// ============================================
// DB_RecipeProgram4 - SpinningCam Program
// Lines: 999
// Generated by SpinningCam  [2026-08-13 21:01:36]
// ============================================
//
// --- MAKINE AYARLARI ---
// Machine Origin  : X=0.0, Z=0.0
// Axis Direction  : X=NORMAL, Z=NORMAL
// Output Mode     : RADIUS
// G54 Offset      : X=0.0, Z=0.0
// Home            : X=-396.641, Z=-174.0
// Retract         : X=-10.0, Z=-10.0
//
// --- PARCA / BLANK ---
// Blank Radius    : 155.0 mm
// Blank Z Shift   : 0.0 mm
// Final Thickness : 0.8 mm
// Min Safety Gap  : 0.0 mm
//
// --- MANDREL POZISYON ---
// Mandrel Offset  : X=0.0, Z=0.0
// Mandrel Rot     : Rx=90.0, Ry=0.0, Rz=0.0
//
// --- OPERASYONLAR ---
// Op1: ROUGHING, 1 paso, T004, R=44.56mm, RPM=800.0, mm_min=800.0
// Op2: ROUGHING, 1 paso, T004, R=44.56mm, RPM=800.0, mm_min=800.0
// Op3: ROUGHING, 1 paso, T004, R=44.56mm, RPM=800.0, mm_min=800.0
// Op4: ROUGHING, 1 paso, T004, R=44.56mm, RPM=800.0, mm_min=800.0
// Op5: ROUGHING, 1 paso, T004, R=44.56mm, RPM=800.0, mm_min=800.0
// Op6: ROUGHING, 1 paso, T004, R=44.56mm, RPM=800.0, mm_min=500.0
// Op7: ROUGHING, 1 paso, T004, R=44.56mm, RPM=800.0, mm_min=500.0
// Op8: ROUGHING, 1 paso, T004, R=44.56mm, RPM=800.0, mm_min=800.0
// Op9: ROUGHING, 1 paso, T004, R=44.56mm, RPM=800.0, mm_min=800.0
// Op10: ROUGHING, 1 paso, T004, R=44.56mm, RPM=800.0, mm_min=800.0
// Op11: ROUGHING, 1 paso, T004, R=44.56mm, RPM=800.0, mm_min=800.0
// Op12: ROUGHING, 1 paso, T004, R=44.56mm, RPM=800.0, mm_min=800.0
// Op13: ROUGHING, 1 paso, T004, R=44.56mm, RPM=800.0, mm_min=400.0
// Op14: ROUGHING, 1 paso, T004, R=44.56mm, RPM=800.0, mm_min=400.0
// Op15: ROUGHING, 1 paso, T004, R=44.56mm, RPM=800.0, mm_min=400.0
// Op16: ROUGHING, 1 paso, T004, R=44.56mm, RPM=800.0, mm_min=400.0
// Op17: ROUGHING, 3 paso, T004, R=44.56mm, RPM=800.0, mm_min=400.0
// Op18: ROUGHING, 3 paso, T004, R=44.56mm, RPM=800.0, mm_min=400.0
// Op19: ROUGHING, 1 paso, T004, R=44.56mm, RPM=800.0, mm_min=800.0
// Op20: ROUGHING, 3 paso, T004, R=44.56mm, RPM=800.0, mm_min=400.0
// Op21: ROUGHING, 3 paso, T004, R=44.56mm, RPM=800.0, mm_min=400.0
// Op22: ROUGHING, 3 paso, T004, R=44.56mm, RPM=800.0, mm_min=400.0
// Op23: ROUGHING, 1 paso, T004, R=44.56mm, RPM=800.0, mm_min=400.0
// Op24: ROUGHING, 3 paso, T004, R=44.56mm, RPM=800.0, mm_min=400.0
// Op25: ROUGHING, 3 paso, T004, R=44.56mm, RPM=800.0, mm_min=400.0
// Op26: ROUGHING, 3 paso, T004, R=44.56mm, RPM=800.0, mm_min=400.0
// Op27: ROUGHING, 3 paso, T004, R=44.56mm, RPM=800.0, mm_min=400.0
// Op28: ROUGHING, 3 paso, T004, R=44.56mm, RPM=800.0, mm_min=400.0
// Op29: ROUGHING, 3 paso, T004, R=44.56mm, RPM=800.0, mm_min=400.0
// Op30: CUTTING, 1 paso, T0102, R=77.53mm, RPM=300.0, mm_min=50.0
// ============================================

DATA_BLOCK "DB_RecipeProgram4"
{ S7_Optimized_Access := 'FALSE' }
VERSION : 0.2
// UNLINKED restored 2026-08-13: the work-memory workaround is withdrawn, the
// chunked loader replaces it. This DB is back in load memory and costs no work
// memory. Its Lines array is declared in CHUNKS (Lines1..Lines10, 100 lines each)
// because READ_DBL can only point at a whole declared member -- see
// tools/split_recipe_db.py, which produced this layout from the CAM export.
UNLINKED
NON_RETAIN
    VAR
        Header : "RecipeHeader";
        Lines1 : Array[0..99] of "RecipeLine"; // global lines 0..99
        Lines2 : Array[0..99] of "RecipeLine"; // global lines 100..199
        Lines3 : Array[0..99] of "RecipeLine"; // global lines 200..299
        Lines4 : Array[0..99] of "RecipeLine"; // global lines 300..399
        Lines5 : Array[0..99] of "RecipeLine"; // global lines 400..499
        Lines6 : Array[0..99] of "RecipeLine"; // global lines 500..599
        Lines7 : Array[0..99] of "RecipeLine"; // global lines 600..699
        Lines8 : Array[0..99] of "RecipeLine"; // global lines 700..799
        Lines9 : Array[0..99] of "RecipeLine"; // global lines 800..899
        Lines10: Array[0..99] of "RecipeLine"; // global lines 900..999
    END_VAR
BEGIN
    // Header
    Header.sName := 'SpinningCam Program';
    Header.LineCount := 999;
    Header.Valid := TRUE;
    Header.PreScanned := FALSE;
    Header.MinX := 0.000;
    Header.MaxX := 275.949;
    Header.MinZ := 0.000;
    Header.MaxZ := 312.533;

    // --- Tool table (CAM-authored) ---
    Header.ProvidesToolConfig := TRUE;
    Header.ToolCount := 3;
    Header.AutoCalcAngles := FALSE;
    Header.ToolCode_List[1] := 4;
    Header.ToolCode_List[2] := 5;
    Header.ToolCode_List[3] := 6;
    Header.ToolCode_List[4] := 0;  // unused
    Header.ToolAngle_List[1] := 0.0;
    Header.ToolAngle_List[2] := 120.0;
    Header.ToolAngle_List[3] := 240.0;
    Header.ToolAngle_List[4] := 360.0;

    // Recipe Lines (999 total)
    Lines1[0].X := 0.000; Lines1[0].Z := 0.000; Lines1[0].F := 0; Lines1[0].CMD := 0; Lines1[0].Param := 0; // G0 Rapid
    Lines1[1].X := 0.000; Lines1[1].Z := 0.000; Lines1[1].F := 0; Lines1[1].CMD := 0; Lines1[1].Param := 0; // G0 Rapid
    Lines1[2].X := 0.000; Lines1[2].Z := 0.000; Lines1[2].F := 0; Lines1[2].CMD := 40; Lines1[2].Param := 80; // Cylinder GOTO 0 mm
    Lines1[3].X := 0.000; Lines1[3].Z := 0.000; Lines1[3].F := 0; Lines1[3].CMD := 10; Lines1[3].Param := 4; // Tool Change T4
    Lines1[4].X := 0.000; Lines1[4].Z := 0.000; Lines1[4].F := 0; Lines1[4].CMD := 20; Lines1[4].Param := 80; // Spindle ON 800 RPM
    Lines1[5].X := 0.000; Lines1[5].Z := 0.000; Lines1[5].F := 0; Lines1[5].CMD := 41; Lines1[5].Param := 1; // M41 (Clamp On) P1 [Op1 P1]
    Lines1[6].X := 275.742; Lines1[6].Z := 181.000; Lines1[6].F := 0; Lines1[6].CMD := 0; Lines1[6].Param := 0; // G0 Rapid [Op1 P1]
    Lines1[7].X := 275.736; Lines1[7].Z := 184.000; Lines1[7].F := 800; Lines1[7].CMD := 1; Lines1[7].Param := 0; // G1 Linear [Op1 P1]
    Lines1[8].X := 188.561; Lines1[8].Z := 203.393; Lines1[8].F := 800; Lines1[8].CMD := 1; Lines1[8].Param := 0; // G1 Linear [Op1 P1]
    Lines1[9].X := 178.561; Lines1[9].Z := 193.393; Lines1[9].F := 0; Lines1[9].CMD := 0; Lines1[9].Param := 0; // G0 Rapid [Op1 P1]
    Lines1[10].X := 178.561; Lines1[10].Z := 193.393; Lines1[10].F := 0; Lines1[10].CMD := 20; Lines1[10].Param := 80; // Spindle ON 800 RPM [Op1 P1]
    Lines1[11].X := 275.742; Lines1[11].Z := 182.538; Lines1[11].F := 0; Lines1[11].CMD := 0; Lines1[11].Param := 0; // G0 Rapid [Op2 P1]
    Lines1[12].X := 275.731; Lines1[12].Z := 185.538; Lines1[12].F := 800; Lines1[12].CMD := 1; Lines1[12].Param := 0; // G1 Linear [Op2 P1]
    Lines1[13].X := 185.741; Lines1[13].Z := 218.401; Lines1[13].F := 800; Lines1[13].CMD := 1; Lines1[13].Param := 0; // G1 Linear [Op2 P1]
    Lines1[14].X := 175.741; Lines1[14].Z := 208.401; Lines1[14].F := 0; Lines1[14].CMD := 0; Lines1[14].Param := 0; // G0 Rapid [Op2 P1]
    Lines1[15].X := 175.741; Lines1[15].Z := 208.401; Lines1[15].F := 0; Lines1[15].CMD := 20; Lines1[15].Param := 80; // Spindle ON 800 RPM [Op2 P1]
    Lines1[16].X := 275.747; Lines1[16].Z := 181.000; Lines1[16].F := 0; Lines1[16].CMD := 0; Lines1[16].Param := 0; // G0 Rapid [Op3 P1]
    Lines1[17].X := 275.718; Lines1[17].Z := 189.000; Lines1[17].F := 800; Lines1[17].CMD := 1; Lines1[17].Param := 0; // G1 Linear [Op3 P1]
    Lines1[18].X := 274.433; Lines1[18].Z := 189.804; Lines1[18].F := 800; Lines1[18].CMD := 1; Lines1[18].Param := 0; // G1 Linear [Op3 P1]
    Lines1[19].X := 273.146; Lines1[19].Z := 190.603; Lines1[19].F := 800; Lines1[19].CMD := 1; Lines1[19].Param := 0; // G1 Linear [Op3 P1]
    Lines1[20].X := 271.856; Lines1[20].Z := 191.396; Lines1[20].F := 800; Lines1[20].CMD := 1; Lines1[20].Param := 0; // G1 Linear [Op3 P1]
    Lines1[21].X := 270.563; Lines1[21].Z := 192.184; Lines1[21].F := 800; Lines1[21].CMD := 1; Lines1[21].Param := 0; // G1 Linear [Op3 P1]
    Lines1[22].X := 269.269; Lines1[22].Z := 192.967; Lines1[22].F := 800; Lines1[22].CMD := 1; Lines1[22].Param := 0; // G1 Linear [Op3 P1]
    Lines1[23].X := 267.971; Lines1[23].Z := 193.745; Lines1[23].F := 800; Lines1[23].CMD := 1; Lines1[23].Param := 0; // G1 Linear [Op3 P1]
    Lines1[24].X := 266.672; Lines1[24].Z := 194.517; Lines1[24].F := 800; Lines1[24].CMD := 1; Lines1[24].Param := 0; // G1 Linear [Op3 P1]
    Lines1[25].X := 265.370; Lines1[25].Z := 195.285; Lines1[25].F := 800; Lines1[25].CMD := 1; Lines1[25].Param := 0; // G1 Linear [Op3 P1]
    Lines1[26].X := 264.065; Lines1[26].Z := 196.047; Lines1[26].F := 800; Lines1[26].CMD := 1; Lines1[26].Param := 0; // G1 Linear [Op3 P1]
    Lines1[27].X := 262.758; Lines1[27].Z := 196.803; Lines1[27].F := 800; Lines1[27].CMD := 1; Lines1[27].Param := 0; // G1 Linear [Op3 P1]
    Lines1[28].X := 261.448; Lines1[28].Z := 197.555; Lines1[28].F := 800; Lines1[28].CMD := 1; Lines1[28].Param := 0; // G1 Linear [Op3 P1]
    Lines1[29].X := 260.136; Lines1[29].Z := 198.301; Lines1[29].F := 800; Lines1[29].CMD := 1; Lines1[29].Param := 0; // G1 Linear [Op3 P1]
    Lines1[30].X := 258.822; Lines1[30].Z := 199.042; Lines1[30].F := 800; Lines1[30].CMD := 1; Lines1[30].Param := 0; // G1 Linear [Op3 P1]
    Lines1[31].X := 257.505; Lines1[31].Z := 199.778; Lines1[31].F := 800; Lines1[31].CMD := 1; Lines1[31].Param := 0; // G1 Linear [Op3 P1]
    Lines1[32].X := 256.186; Lines1[32].Z := 200.508; Lines1[32].F := 800; Lines1[32].CMD := 1; Lines1[32].Param := 0; // G1 Linear [Op3 P1]
    Lines1[33].X := 254.864; Lines1[33].Z := 201.233; Lines1[33].F := 800; Lines1[33].CMD := 1; Lines1[33].Param := 0; // G1 Linear [Op3 P1]
    Lines1[34].X := 253.540; Lines1[34].Z := 201.953; Lines1[34].F := 800; Lines1[34].CMD := 1; Lines1[34].Param := 0; // G1 Linear [Op3 P1]
    Lines1[35].X := 252.213; Lines1[35].Z := 202.668; Lines1[35].F := 800; Lines1[35].CMD := 1; Lines1[35].Param := 0; // G1 Linear [Op3 P1]
    Lines1[36].X := 250.884; Lines1[36].Z := 203.377; Lines1[36].F := 800; Lines1[36].CMD := 1; Lines1[36].Param := 0; // G1 Linear [Op3 P1]
    Lines1[37].X := 249.552; Lines1[37].Z := 204.081; Lines1[37].F := 800; Lines1[37].CMD := 1; Lines1[37].Param := 0; // G1 Linear [Op3 P1]
    Lines1[38].X := 248.218; Lines1[38].Z := 204.780; Lines1[38].F := 800; Lines1[38].CMD := 1; Lines1[38].Param := 0; // G1 Linear [Op3 P1]
    Lines1[39].X := 246.881; Lines1[39].Z := 205.474; Lines1[39].F := 800; Lines1[39].CMD := 1; Lines1[39].Param := 0; // G1 Linear [Op3 P1]
    Lines1[40].X := 245.542; Lines1[40].Z := 206.162; Lines1[40].F := 800; Lines1[40].CMD := 1; Lines1[40].Param := 0; // G1 Linear [Op3 P1]
    Lines1[41].X := 244.201; Lines1[41].Z := 206.846; Lines1[41].F := 800; Lines1[41].CMD := 1; Lines1[41].Param := 0; // G1 Linear [Op3 P1]
    Lines1[42].X := 242.633; Lines1[42].Z := 207.636; Lines1[42].F := 800; Lines1[42].CMD := 1; Lines1[42].Param := 0; // G1 Linear [Op3 P1]
    Lines1[43].X := 241.286; Lines1[43].Z := 208.308; Lines1[43].F := 800; Lines1[43].CMD := 1; Lines1[43].Param := 0; // G1 Linear [Op3 P1]
    Lines1[44].X := 239.937; Lines1[44].Z := 208.974; Lines1[44].F := 800; Lines1[44].CMD := 1; Lines1[44].Param := 0; // G1 Linear [Op3 P1]
    Lines1[45].X := 238.585; Lines1[45].Z := 209.636; Lines1[45].F := 800; Lines1[45].CMD := 1; Lines1[45].Param := 0; // G1 Linear [Op3 P1]
    Lines1[46].X := 237.231; Lines1[46].Z := 210.292; Lines1[46].F := 800; Lines1[46].CMD := 1; Lines1[46].Param := 0; // G1 Linear [Op3 P1]
    Lines1[47].X := 235.874; Lines1[47].Z := 210.942; Lines1[47].F := 800; Lines1[47].CMD := 1; Lines1[47].Param := 0; // G1 Linear [Op3 P1]
    Lines1[48].X := 234.515; Lines1[48].Z := 211.588; Lines1[48].F := 800; Lines1[48].CMD := 1; Lines1[48].Param := 0; // G1 Linear [Op3 P1]
    Lines1[49].X := 233.154; Lines1[49].Z := 212.228; Lines1[49].F := 800; Lines1[49].CMD := 1; Lines1[49].Param := 0; // G1 Linear [Op3 P1]
    Lines1[50].X := 231.562; Lines1[50].Z := 212.969; Lines1[50].F := 800; Lines1[50].CMD := 1; Lines1[50].Param := 0; // G1 Linear [Op3 P1]
    Lines1[51].X := 230.195; Lines1[51].Z := 213.597; Lines1[51].F := 800; Lines1[51].CMD := 1; Lines1[51].Param := 0; // G1 Linear [Op3 P1]
    Lines1[52].X := 228.826; Lines1[52].Z := 214.221; Lines1[52].F := 800; Lines1[52].CMD := 1; Lines1[52].Param := 0; // G1 Linear [Op3 P1]
    Lines1[53].X := 227.454; Lines1[53].Z := 214.839; Lines1[53].F := 800; Lines1[53].CMD := 1; Lines1[53].Param := 0; // G1 Linear [Op3 P1]
    Lines1[54].X := 226.080; Lines1[54].Z := 215.453; Lines1[54].F := 800; Lines1[54].CMD := 1; Lines1[54].Param := 0; // G1 Linear [Op3 P1]
    Lines1[55].X := 224.703; Lines1[55].Z := 216.060; Lines1[55].F := 800; Lines1[55].CMD := 1; Lines1[55].Param := 0; // G1 Linear [Op3 P1]
    Lines1[56].X := 223.324; Lines1[56].Z := 216.663; Lines1[56].F := 800; Lines1[56].CMD := 1; Lines1[56].Param := 0; // G1 Linear [Op3 P1]
    Lines1[57].X := 221.942; Lines1[57].Z := 217.260; Lines1[57].F := 800; Lines1[57].CMD := 1; Lines1[57].Param := 0; // G1 Linear [Op3 P1]
    Lines1[58].X := 220.558; Lines1[58].Z := 217.853; Lines1[58].F := 800; Lines1[58].CMD := 1; Lines1[58].Param := 0; // G1 Linear [Op3 P1]
    Lines1[59].X := 219.172; Lines1[59].Z := 218.439; Lines1[59].F := 800; Lines1[59].CMD := 1; Lines1[59].Param := 0; // G1 Linear [Op3 P1]
    Lines1[60].X := 217.783; Lines1[60].Z := 219.021; Lines1[60].F := 800; Lines1[60].CMD := 1; Lines1[60].Param := 0; // G1 Linear [Op3 P1]
    Lines1[61].X := 216.391; Lines1[61].Z := 219.597; Lines1[61].F := 800; Lines1[61].CMD := 1; Lines1[61].Param := 0; // G1 Linear [Op3 P1]
    Lines1[62].X := 214.997; Lines1[62].Z := 220.169; Lines1[62].F := 800; Lines1[62].CMD := 1; Lines1[62].Param := 0; // G1 Linear [Op3 P1]
    Lines1[63].X := 213.601; Lines1[63].Z := 220.734; Lines1[63].F := 800; Lines1[63].CMD := 1; Lines1[63].Param := 0; // G1 Linear [Op3 P1]
    Lines1[64].X := 212.202; Lines1[64].Z := 221.295; Lines1[64].F := 800; Lines1[64].CMD := 1; Lines1[64].Param := 0; // G1 Linear [Op3 P1]
    Lines1[65].X := 210.801; Lines1[65].Z := 221.850; Lines1[65].F := 800; Lines1[65].CMD := 1; Lines1[65].Param := 0; // G1 Linear [Op3 P1]
    Lines1[66].X := 209.397; Lines1[66].Z := 222.401; Lines1[66].F := 800; Lines1[66].CMD := 1; Lines1[66].Param := 0; // G1 Linear [Op3 P1]
    Lines1[67].X := 207.991; Lines1[67].Z := 222.945; Lines1[67].F := 800; Lines1[67].CMD := 1; Lines1[67].Param := 0; // G1 Linear [Op3 P1]
    Lines1[68].X := 206.582; Lines1[68].Z := 223.485; Lines1[68].F := 800; Lines1[68].CMD := 1; Lines1[68].Param := 0; // G1 Linear [Op3 P1]
    Lines1[69].X := 205.171; Lines1[69].Z := 224.019; Lines1[69].F := 800; Lines1[69].CMD := 1; Lines1[69].Param := 0; // G1 Linear [Op3 P1]
    Lines1[70].X := 203.758; Lines1[70].Z := 224.548; Lines1[70].F := 800; Lines1[70].CMD := 1; Lines1[70].Param := 0; // G1 Linear [Op3 P1]
    Lines1[71].X := 202.342; Lines1[71].Z := 225.072; Lines1[71].F := 800; Lines1[71].CMD := 1; Lines1[71].Param := 0; // G1 Linear [Op3 P1]
    Lines1[72].X := 200.923; Lines1[72].Z := 225.591; Lines1[72].F := 800; Lines1[72].CMD := 1; Lines1[72].Param := 0; // G1 Linear [Op3 P1]
    Lines1[73].X := 199.502; Lines1[73].Z := 226.104; Lines1[73].F := 800; Lines1[73].CMD := 1; Lines1[73].Param := 0; // G1 Linear [Op3 P1]
    Lines1[74].X := 198.079; Lines1[74].Z := 226.612; Lines1[74].F := 800; Lines1[74].CMD := 1; Lines1[74].Param := 0; // G1 Linear [Op3 P1]
    Lines1[75].X := 196.653; Lines1[75].Z := 227.115; Lines1[75].F := 800; Lines1[75].CMD := 1; Lines1[75].Param := 0; // G1 Linear [Op3 P1]
    Lines1[76].X := 195.225; Lines1[76].Z := 227.613; Lines1[76].F := 800; Lines1[76].CMD := 1; Lines1[76].Param := 0; // G1 Linear [Op3 P1]
    Lines1[77].X := 193.794; Lines1[77].Z := 228.105; Lines1[77].F := 800; Lines1[77].CMD := 1; Lines1[77].Param := 0; // G1 Linear [Op3 P1]
    Lines1[78].X := 192.361; Lines1[78].Z := 228.592; Lines1[78].F := 800; Lines1[78].CMD := 1; Lines1[78].Param := 0; // G1 Linear [Op3 P1]
    Lines1[79].X := 190.925; Lines1[79].Z := 229.074; Lines1[79].F := 800; Lines1[79].CMD := 1; Lines1[79].Param := 0; // G1 Linear [Op3 P1]
    Lines1[80].X := 189.487; Lines1[80].Z := 229.551; Lines1[80].F := 800; Lines1[80].CMD := 1; Lines1[80].Param := 0; // G1 Linear [Op3 P1]
    Lines1[81].X := 188.046; Lines1[81].Z := 230.022; Lines1[81].F := 800; Lines1[81].CMD := 1; Lines1[81].Param := 0; // G1 Linear [Op3 P1]
    Lines1[82].X := 178.046; Lines1[82].Z := 220.022; Lines1[82].F := 0; Lines1[82].CMD := 0; Lines1[82].Param := 0; // G0 Rapid [Op3 P1]
    Lines1[83].X := 178.046; Lines1[83].Z := 220.022; Lines1[83].F := 0; Lines1[83].CMD := 20; Lines1[83].Param := 80; // Spindle ON 800 RPM [Op3 P1]
    Lines1[84].X := 275.747; Lines1[84].Z := 181.000; Lines1[84].F := 0; Lines1[84].CMD := 0; Lines1[84].Param := 0; // G0 Rapid [Op4 P1]
    Lines1[85].X := 275.703; Lines1[85].Z := 193.000; Lines1[85].F := 800; Lines1[85].CMD := 1; Lines1[85].Param := 0; // G1 Linear [Op4 P1]
    Lines1[86].X := 274.461; Lines1[86].Z := 193.867; Lines1[86].F := 800; Lines1[86].CMD := 1; Lines1[86].Param := 0; // G1 Linear [Op4 P1]
    Lines1[87].X := 273.215; Lines1[87].Z := 194.728; Lines1[87].F := 800; Lines1[87].CMD := 1; Lines1[87].Param := 0; // G1 Linear [Op4 P1]
    Lines1[88].X := 271.967; Lines1[88].Z := 195.585; Lines1[88].F := 800; Lines1[88].CMD := 1; Lines1[88].Param := 0; // G1 Linear [Op4 P1]
    Lines1[89].X := 270.508; Lines1[89].Z := 196.578; Lines1[89].F := 800; Lines1[89].CMD := 1; Lines1[89].Param := 0; // G1 Linear [Op4 P1]
    Lines1[90].X := 269.254; Lines1[90].Z := 197.425; Lines1[90].F := 800; Lines1[90].CMD := 1; Lines1[90].Param := 0; // G1 Linear [Op4 P1]
    Lines1[91].X := 267.998; Lines1[91].Z := 198.266; Lines1[91].F := 800; Lines1[91].CMD := 1; Lines1[91].Param := 0; // G1 Linear [Op4 P1]
    Lines1[92].X := 266.529; Lines1[92].Z := 199.241; Lines1[92].F := 800; Lines1[92].CMD := 1; Lines1[92].Param := 0; // G1 Linear [Op4 P1]
    Lines1[93].X := 265.267; Lines1[93].Z := 200.072; Lines1[93].F := 800; Lines1[93].CMD := 1; Lines1[93].Param := 0; // G1 Linear [Op4 P1]
    Lines1[94].X := 264.002; Lines1[94].Z := 200.898; Lines1[94].F := 800; Lines1[94].CMD := 1; Lines1[94].Param := 0; // G1 Linear [Op4 P1]
    Lines1[95].X := 262.735; Lines1[95].Z := 201.719; Lines1[95].F := 800; Lines1[95].CMD := 1; Lines1[95].Param := 0; // G1 Linear [Op4 P1]
    Lines1[96].X := 261.254; Lines1[96].Z := 202.670; Lines1[96].F := 800; Lines1[96].CMD := 1; Lines1[96].Param := 0; // G1 Linear [Op4 P1]
    Lines1[97].X := 259.981; Lines1[97].Z := 203.481; Lines1[97].F := 800; Lines1[97].CMD := 1; Lines1[97].Param := 0; // G1 Linear [Op4 P1]
    Lines1[98].X := 258.705; Lines1[98].Z := 204.286; Lines1[98].F := 800; Lines1[98].CMD := 1; Lines1[98].Param := 0; // G1 Linear [Op4 P1]
    Lines1[99].X := 257.427; Lines1[99].Z := 205.087; Lines1[99].F := 800; Lines1[99].CMD := 1; Lines1[99].Param := 0; // G1 Linear [Op4 P1]
    Lines2[0].X := 256.147; Lines2[0].Z := 205.882; Lines2[0].F := 800; Lines2[0].CMD := 1; Lines2[0].Param := 0; // G1 Linear [Op4 P1]
    Lines2[1].X := 254.864; Lines2[1].Z := 206.673; Lines2[1].F := 800; Lines2[1].CMD := 1; Lines2[1].Param := 0; // G1 Linear [Op4 P1]
    Lines2[2].X := 253.578; Lines2[2].Z := 207.459; Lines2[2].F := 800; Lines2[2].CMD := 1; Lines2[2].Param := 0; // G1 Linear [Op4 P1]
    Lines2[3].X := 252.074; Lines2[3].Z := 208.370; Lines2[3].F := 800; Lines2[3].CMD := 1; Lines2[3].Param := 0; // G1 Linear [Op4 P1]
    Lines2[4].X := 250.783; Lines2[4].Z := 209.145; Lines2[4].F := 800; Lines2[4].CMD := 1; Lines2[4].Param := 0; // G1 Linear [Op4 P1]
    Lines2[5].X := 249.489; Lines2[5].Z := 209.916; Lines2[5].F := 800; Lines2[5].CMD := 1; Lines2[5].Param := 0; // G1 Linear [Op4 P1]
    Lines2[6].X := 248.192; Lines2[6].Z := 210.681; Lines2[6].F := 800; Lines2[6].CMD := 1; Lines2[6].Param := 0; // G1 Linear [Op4 P1]
    Lines2[7].X := 246.676; Lines2[7].Z := 211.568; Lines2[7].F := 800; Lines2[7].CMD := 1; Lines2[7].Param := 0; // G1 Linear [Op4 P1]
    Lines2[8].X := 245.374; Lines2[8].Z := 212.323; Lines2[8].F := 800; Lines2[8].CMD := 1; Lines2[8].Param := 0; // G1 Linear [Op4 P1]
    Lines2[9].X := 244.069; Lines2[9].Z := 213.073; Lines2[9].F := 800; Lines2[9].CMD := 1; Lines2[9].Param := 0; // G1 Linear [Op4 P1]
    Lines2[10].X := 242.761; Lines2[10].Z := 213.819; Lines2[10].F := 800; Lines2[10].CMD := 1; Lines2[10].Param := 0; // G1 Linear [Op4 P1]
    Lines2[11].X := 241.451; Lines2[11].Z := 214.559; Lines2[11].F := 800; Lines2[11].CMD := 1; Lines2[11].Param := 0; // G1 Linear [Op4 P1]
    Lines2[12].X := 239.919; Lines2[12].Z := 215.417; Lines2[12].F := 800; Lines2[12].CMD := 1; Lines2[12].Param := 0; // G1 Linear [Op4 P1]
    Lines2[13].X := 238.603; Lines2[13].Z := 216.146; Lines2[13].F := 800; Lines2[13].CMD := 1; Lines2[13].Param := 0; // G1 Linear [Op4 P1]
    Lines2[14].X := 237.285; Lines2[14].Z := 216.871; Lines2[14].F := 800; Lines2[14].CMD := 1; Lines2[14].Param := 0; // G1 Linear [Op4 P1]
    Lines2[15].X := 235.964; Lines2[15].Z := 217.591; Lines2[15].F := 800; Lines2[15].CMD := 1; Lines2[15].Param := 0; // G1 Linear [Op4 P1]
    Lines2[16].X := 234.640; Lines2[16].Z := 218.306; Lines2[16].F := 800; Lines2[16].CMD := 1; Lines2[16].Param := 0; // G1 Linear [Op4 P1]
    Lines2[17].X := 233.314; Lines2[17].Z := 219.017; Lines2[17].F := 800; Lines2[17].CMD := 1; Lines2[17].Param := 0; // G1 Linear [Op4 P1]
    Lines2[18].X := 231.985; Lines2[18].Z := 219.722; Lines2[18].F := 800; Lines2[18].CMD := 1; Lines2[18].Param := 0; // G1 Linear [Op4 P1]
    Lines2[19].X := 230.654; Lines2[19].Z := 220.422; Lines2[19].F := 800; Lines2[19].CMD := 1; Lines2[19].Param := 0; // G1 Linear [Op4 P1]
    Lines2[20].X := 229.320; Lines2[20].Z := 221.118; Lines2[20].F := 800; Lines2[20].CMD := 1; Lines2[20].Param := 0; // G1 Linear [Op4 P1]
    Lines2[21].X := 227.760; Lines2[21].Z := 221.923; Lines2[21].F := 800; Lines2[21].CMD := 1; Lines2[21].Param := 0; // G1 Linear [Op4 P1]
    Lines2[22].X := 226.420; Lines2[22].Z := 222.608; Lines2[22].F := 800; Lines2[22].CMD := 1; Lines2[22].Param := 0; // G1 Linear [Op4 P1]
    Lines2[23].X := 225.078; Lines2[23].Z := 223.288; Lines2[23].F := 800; Lines2[23].CMD := 1; Lines2[23].Param := 0; // G1 Linear [Op4 P1]
    Lines2[24].X := 223.733; Lines2[24].Z := 223.963; Lines2[24].F := 800; Lines2[24].CMD := 1; Lines2[24].Param := 0; // G1 Linear [Op4 P1]
    Lines2[25].X := 222.386; Lines2[25].Z := 224.634; Lines2[25].F := 800; Lines2[25].CMD := 1; Lines2[25].Param := 0; // G1 Linear [Op4 P1]
    Lines2[26].X := 221.035; Lines2[26].Z := 225.299; Lines2[26].F := 800; Lines2[26].CMD := 1; Lines2[26].Param := 0; // G1 Linear [Op4 P1]
    Lines2[27].X := 219.683; Lines2[27].Z := 225.960; Lines2[27].F := 800; Lines2[27].CMD := 1; Lines2[27].Param := 0; // G1 Linear [Op4 P1]
    Lines2[28].X := 218.327; Lines2[28].Z := 226.615; Lines2[28].F := 800; Lines2[28].CMD := 1; Lines2[28].Param := 0; // G1 Linear [Op4 P1]
    Lines2[29].X := 216.969; Lines2[29].Z := 227.266; Lines2[29].F := 800; Lines2[29].CMD := 1; Lines2[29].Param := 0; // G1 Linear [Op4 P1]
    Lines2[30].X := 215.609; Lines2[30].Z := 227.912; Lines2[30].F := 800; Lines2[30].CMD := 1; Lines2[30].Param := 0; // G1 Linear [Op4 P1]
    Lines2[31].X := 214.018; Lines2[31].Z := 228.659; Lines2[31].F := 800; Lines2[31].CMD := 1; Lines2[31].Param := 0; // G1 Linear [Op4 P1]
    Lines2[32].X := 212.652; Lines2[32].Z := 229.295; Lines2[32].F := 800; Lines2[32].CMD := 1; Lines2[32].Param := 0; // G1 Linear [Op4 P1]
    Lines2[33].X := 211.283; Lines2[33].Z := 229.925; Lines2[33].F := 800; Lines2[33].CMD := 1; Lines2[33].Param := 0; // G1 Linear [Op4 P1]
    Lines2[34].X := 209.912; Lines2[34].Z := 230.550; Lines2[34].F := 800; Lines2[34].CMD := 1; Lines2[34].Param := 0; // G1 Linear [Op4 P1]
    Lines2[35].X := 208.538; Lines2[35].Z := 231.171; Lines2[35].F := 800; Lines2[35].CMD := 1; Lines2[35].Param := 0; // G1 Linear [Op4 P1]
    Lines2[36].X := 207.161; Lines2[36].Z := 231.787; Lines2[36].F := 800; Lines2[36].CMD := 1; Lines2[36].Param := 0; // G1 Linear [Op4 P1]
    Lines2[37].X := 205.782; Lines2[37].Z := 232.398; Lines2[37].F := 800; Lines2[37].CMD := 1; Lines2[37].Param := 0; // G1 Linear [Op4 P1]
    Lines2[38].X := 204.400; Lines2[38].Z := 233.004; Lines2[38].F := 800; Lines2[38].CMD := 1; Lines2[38].Param := 0; // G1 Linear [Op4 P1]
    Lines2[39].X := 202.785; Lines2[39].Z := 233.705; Lines2[39].F := 800; Lines2[39].CMD := 1; Lines2[39].Param := 0; // G1 Linear [Op4 P1]
    Lines2[40].X := 201.397; Lines2[40].Z := 234.300; Lines2[40].F := 800; Lines2[40].CMD := 1; Lines2[40].Param := 0; // G1 Linear [Op4 P1]
    Lines2[41].X := 200.007; Lines2[41].Z := 234.890; Lines2[41].F := 800; Lines2[41].CMD := 1; Lines2[41].Param := 0; // G1 Linear [Op4 P1]
    Lines2[42].X := 198.614; Lines2[42].Z := 235.476; Lines2[42].F := 800; Lines2[42].CMD := 1; Lines2[42].Param := 0; // G1 Linear [Op4 P1]
    Lines2[43].X := 196.986; Lines2[43].Z := 236.153; Lines2[43].F := 800; Lines2[43].CMD := 1; Lines2[43].Param := 0; // G1 Linear [Op4 P1]
    Lines2[44].X := 195.588; Lines2[44].Z := 236.728; Lines2[44].F := 800; Lines2[44].CMD := 1; Lines2[44].Param := 0; // G1 Linear [Op4 P1]
    Lines2[45].X := 194.187; Lines2[45].Z := 237.298; Lines2[45].F := 800; Lines2[45].CMD := 1; Lines2[45].Param := 0; // G1 Linear [Op4 P1]
    Lines2[46].X := 192.783; Lines2[46].Z := 237.864; Lines2[46].F := 800; Lines2[46].CMD := 1; Lines2[46].Param := 0; // G1 Linear [Op4 P1]
    Lines2[47].X := 191.377; Lines2[47].Z := 238.424; Lines2[47].F := 800; Lines2[47].CMD := 1; Lines2[47].Param := 0; // G1 Linear [Op4 P1]
    Lines2[48].X := 189.733; Lines2[48].Z := 239.072; Lines2[48].F := 800; Lines2[48].CMD := 1; Lines2[48].Param := 0; // G1 Linear [Op4 P1]
    Lines2[49].X := 188.321; Lines2[49].Z := 239.621; Lines2[49].F := 800; Lines2[49].CMD := 1; Lines2[49].Param := 0; // G1 Linear [Op4 P1]
    Lines2[50].X := 178.321; Lines2[50].Z := 229.621; Lines2[50].F := 0; Lines2[50].CMD := 0; Lines2[50].Param := 0; // G0 Rapid [Op4 P1]
    Lines2[51].X := 178.321; Lines2[51].Z := 229.621; Lines2[51].F := 0; Lines2[51].CMD := 20; Lines2[51].Param := 80; // Spindle ON 800 RPM [Op4 P1]
    Lines2[52].X := 275.447; Lines2[52].Z := 181.000; Lines2[52].F := 0; Lines2[52].CMD := 0; Lines2[52].Param := 0; // G0 Rapid [Op5 P1]
    Lines2[53].X := 275.389; Lines2[53].Z := 197.000; Lines2[53].F := 800; Lines2[53].CMD := 1; Lines2[53].Param := 0; // G1 Linear [Op5 P1]
    Lines2[54].X := 274.227; Lines2[54].Z := 197.972; Lines2[54].F := 800; Lines2[54].CMD := 1; Lines2[54].Param := 0; // G1 Linear [Op5 P1]
    Lines2[55].X := 273.062; Lines2[55].Z := 198.939; Lines2[55].F := 800; Lines2[55].CMD := 1; Lines2[55].Param := 0; // G1 Linear [Op5 P1]
    Lines2[56].X := 271.699; Lines2[56].Z := 200.062; Lines2[56].F := 800; Lines2[56].CMD := 1; Lines2[56].Param := 0; // G1 Linear [Op5 P1]
    Lines2[57].X := 270.528; Lines2[57].Z := 201.020; Lines2[57].F := 800; Lines2[57].CMD := 1; Lines2[57].Param := 0; // G1 Linear [Op5 P1]
    Lines2[58].X := 269.353; Lines2[58].Z := 201.973; Lines2[58].F := 800; Lines2[58].CMD := 1; Lines2[58].Param := 0; // G1 Linear [Op5 P1]
    Lines2[59].X := 267.980; Lines2[59].Z := 203.079; Lines2[59].F := 800; Lines2[59].CMD := 1; Lines2[59].Param := 0; // G1 Linear [Op5 P1]
    Lines2[60].X := 266.799; Lines2[60].Z := 204.022; Lines2[60].F := 800; Lines2[60].CMD := 1; Lines2[60].Param := 0; // G1 Linear [Op5 P1]
    Lines2[61].X := 265.615; Lines2[61].Z := 204.961; Lines2[61].F := 800; Lines2[61].CMD := 1; Lines2[61].Param := 0; // G1 Linear [Op5 P1]
    Lines2[62].X := 264.428; Lines2[62].Z := 205.895; Lines2[62].F := 800; Lines2[62].CMD := 1; Lines2[62].Param := 0; // G1 Linear [Op5 P1]
    Lines2[63].X := 263.239; Lines2[63].Z := 206.825; Lines2[63].F := 800; Lines2[63].CMD := 1; Lines2[63].Param := 0; // G1 Linear [Op5 P1]
    Lines2[64].X := 262.046; Lines2[64].Z := 207.750; Lines2[64].F := 800; Lines2[64].CMD := 1; Lines2[64].Param := 0; // G1 Linear [Op5 P1]
    Lines2[65].X := 260.651; Lines2[65].Z := 208.824; Lines2[65].F := 800; Lines2[65].CMD := 1; Lines2[65].Param := 0; // G1 Linear [Op5 P1]
    Lines2[66].X := 259.252; Lines2[66].Z := 209.891; Lines2[66].F := 800; Lines2[66].CMD := 1; Lines2[66].Param := 0; // G1 Linear [Op5 P1]
    Lines2[67].X := 258.050; Lines2[67].Z := 210.801; Lines2[67].F := 800; Lines2[67].CMD := 1; Lines2[67].Param := 0; // G1 Linear [Op5 P1]
    Lines2[68].X := 256.844; Lines2[68].Z := 211.707; Lines2[68].F := 800; Lines2[68].CMD := 1; Lines2[68].Param := 0; // G1 Linear [Op5 P1]
    Lines2[69].X := 255.636; Lines2[69].Z := 212.608; Lines2[69].F := 800; Lines2[69].CMD := 1; Lines2[69].Param := 0; // G1 Linear [Op5 P1]
    Lines2[70].X := 254.425; Lines2[70].Z := 213.504; Lines2[70].F := 800; Lines2[70].CMD := 1; Lines2[70].Param := 0; // G1 Linear [Op5 P1]
    Lines2[71].X := 253.211; Lines2[71].Z := 214.396; Lines2[71].F := 800; Lines2[71].CMD := 1; Lines2[71].Param := 0; // G1 Linear [Op5 P1]
    Lines2[72].X := 251.993; Lines2[72].Z := 215.284; Lines2[72].F := 800; Lines2[72].CMD := 1; Lines2[72].Param := 0; // G1 Linear [Op5 P1]
    Lines2[73].X := 250.570; Lines2[73].Z := 216.314; Lines2[73].F := 800; Lines2[73].CMD := 1; Lines2[73].Param := 0; // G1 Linear [Op5 P1]
    Lines2[74].X := 249.346; Lines2[74].Z := 217.191; Lines2[74].F := 800; Lines2[74].CMD := 1; Lines2[74].Param := 0; // G1 Linear [Op5 P1]
    Lines2[75].X := 248.119; Lines2[75].Z := 218.065; Lines2[75].F := 800; Lines2[75].CMD := 1; Lines2[75].Param := 0; // G1 Linear [Op5 P1]
    Lines2[76].X := 246.685; Lines2[76].Z := 219.078; Lines2[76].F := 800; Lines2[76].CMD := 1; Lines2[76].Param := 0; // G1 Linear [Op5 P1]
    Lines2[77].X := 245.452; Lines2[77].Z := 219.941; Lines2[77].F := 800; Lines2[77].CMD := 1; Lines2[77].Param := 0; // G1 Linear [Op5 P1]
    Lines2[78].X := 244.216; Lines2[78].Z := 220.800; Lines2[78].F := 800; Lines2[78].CMD := 1; Lines2[78].Param := 0; // G1 Linear [Op5 P1]
    Lines2[79].X := 242.977; Lines2[79].Z := 221.654; Lines2[79].F := 800; Lines2[79].CMD := 1; Lines2[79].Param := 0; // G1 Linear [Op5 P1]
    Lines2[80].X := 241.528; Lines2[80].Z := 222.645; Lines2[80].F := 800; Lines2[80].CMD := 1; Lines2[80].Param := 0; // G1 Linear [Op5 P1]
    Lines2[81].X := 240.283; Lines2[81].Z := 223.490; Lines2[81].F := 800; Lines2[81].CMD := 1; Lines2[81].Param := 0; // G1 Linear [Op5 P1]
    Lines2[82].X := 239.034; Lines2[82].Z := 224.330; Lines2[82].F := 800; Lines2[82].CMD := 1; Lines2[82].Param := 0; // G1 Linear [Op5 P1]
    Lines2[83].X := 237.783; Lines2[83].Z := 225.165; Lines2[83].F := 800; Lines2[83].CMD := 1; Lines2[83].Param := 0; // G1 Linear [Op5 P1]
    Lines2[84].X := 236.320; Lines2[84].Z := 226.135; Lines2[84].F := 800; Lines2[84].CMD := 1; Lines2[84].Param := 0; // G1 Linear [Op5 P1]
    Lines2[85].X := 235.062; Lines2[85].Z := 226.960; Lines2[85].F := 800; Lines2[85].CMD := 1; Lines2[85].Param := 0; // G1 Linear [Op5 P1]
    Lines2[86].X := 233.802; Lines2[86].Z := 227.782; Lines2[86].F := 800; Lines2[86].CMD := 1; Lines2[86].Param := 0; // G1 Linear [Op5 P1]
    Lines2[87].X := 232.538; Lines2[87].Z := 228.598; Lines2[87].F := 800; Lines2[87].CMD := 1; Lines2[87].Param := 0; // G1 Linear [Op5 P1]
    Lines2[88].X := 231.272; Lines2[88].Z := 229.410; Lines2[88].F := 800; Lines2[88].CMD := 1; Lines2[88].Param := 0; // G1 Linear [Op5 P1]
    Lines2[89].X := 229.791; Lines2[89].Z := 230.352; Lines2[89].F := 800; Lines2[89].CMD := 1; Lines2[89].Param := 0; // G1 Linear [Op5 P1]
    Lines2[90].X := 228.518; Lines2[90].Z := 231.155; Lines2[90].F := 800; Lines2[90].CMD := 1; Lines2[90].Param := 0; // G1 Linear [Op5 P1]
    Lines2[91].X := 227.242; Lines2[91].Z := 231.953; Lines2[91].F := 800; Lines2[91].CMD := 1; Lines2[91].Param := 0; // G1 Linear [Op5 P1]
    Lines2[92].X := 225.963; Lines2[92].Z := 232.746; Lines2[92].F := 800; Lines2[92].CMD := 1; Lines2[92].Param := 0; // G1 Linear [Op5 P1]
    Lines2[93].X := 224.467; Lines2[93].Z := 233.666; Lines2[93].F := 800; Lines2[93].CMD := 1; Lines2[93].Param := 0; // G1 Linear [Op5 P1]
    Lines2[94].X := 223.182; Lines2[94].Z := 234.449; Lines2[94].F := 800; Lines2[94].CMD := 1; Lines2[94].Param := 0; // G1 Linear [Op5 P1]
    Lines2[95].X := 221.894; Lines2[95].Z := 235.228; Lines2[95].F := 800; Lines2[95].CMD := 1; Lines2[95].Param := 0; // G1 Linear [Op5 P1]
    Lines2[96].X := 220.603; Lines2[96].Z := 236.003; Lines2[96].F := 800; Lines2[96].CMD := 1; Lines2[96].Param := 0; // G1 Linear [Op5 P1]
    Lines2[97].X := 219.093; Lines2[97].Z := 236.901; Lines2[97].F := 800; Lines2[97].CMD := 1; Lines2[97].Param := 0; // G1 Linear [Op5 P1]
    Lines2[98].X := 217.796; Lines2[98].Z := 237.666; Lines2[98].F := 800; Lines2[98].CMD := 1; Lines2[98].Param := 0; // G1 Linear [Op5 P1]
    Lines2[99].X := 216.495; Lines2[99].Z := 238.426; Lines2[99].F := 800; Lines2[99].CMD := 1; Lines2[99].Param := 0; // G1 Linear [Op5 P1]
    Lines3[0].X := 215.192; Lines3[0].Z := 239.181; Lines3[0].F := 800; Lines3[0].CMD := 1; Lines3[0].Param := 0; // G1 Linear [Op5 P1]
    Lines3[1].X := 213.667; Lines3[1].Z := 240.057; Lines3[1].F := 800; Lines3[1].CMD := 1; Lines3[1].Param := 0; // G1 Linear [Op5 P1]
    Lines3[2].X := 212.358; Lines3[2].Z := 240.803; Lines3[2].F := 800; Lines3[2].CMD := 1; Lines3[2].Param := 0; // G1 Linear [Op5 P1]
    Lines3[3].X := 211.045; Lines3[3].Z := 241.545; Lines3[3].F := 800; Lines3[3].CMD := 1; Lines3[3].Param := 0; // G1 Linear [Op5 P1]
    Lines3[4].X := 209.729; Lines3[4].Z := 242.282; Lines3[4].F := 800; Lines3[4].CMD := 1; Lines3[4].Param := 0; // G1 Linear [Op5 P1]
    Lines3[5].X := 208.190; Lines3[5].Z := 243.136; Lines3[5].F := 800; Lines3[5].CMD := 1; Lines3[5].Param := 0; // G1 Linear [Op5 P1]
    Lines3[6].X := 206.868; Lines3[6].Z := 243.863; Lines3[6].F := 800; Lines3[6].CMD := 1; Lines3[6].Param := 0; // G1 Linear [Op5 P1]
    Lines3[7].X := 205.322; Lines3[7].Z := 244.705; Lines3[7].F := 800; Lines3[7].CMD := 1; Lines3[7].Param := 0; // G1 Linear [Op5 P1]
    Lines3[8].X := 203.994; Lines3[8].Z := 245.422; Lines3[8].F := 800; Lines3[8].CMD := 1; Lines3[8].Param := 0; // G1 Linear [Op5 P1]
    Lines3[9].X := 202.662; Lines3[9].Z := 246.135; Lines3[9].F := 800; Lines3[9].CMD := 1; Lines3[9].Param := 0; // G1 Linear [Op5 P1]
    Lines3[10].X := 201.328; Lines3[10].Z := 246.844; Lines3[10].F := 800; Lines3[10].CMD := 1; Lines3[10].Param := 0; // G1 Linear [Op5 P1]
    Lines3[11].X := 199.990; Lines3[11].Z := 247.547; Lines3[11].F := 800; Lines3[11].CMD := 1; Lines3[11].Param := 0; // G1 Linear [Op5 P1]
    Lines3[12].X := 198.650; Lines3[12].Z := 248.246; Lines3[12].F := 800; Lines3[12].CMD := 1; Lines3[12].Param := 0; // G1 Linear [Op5 P1]
    Lines3[13].X := 197.082; Lines3[13].Z := 249.056; Lines3[13].F := 800; Lines3[13].CMD := 1; Lines3[13].Param := 0; // G1 Linear [Op5 P1]
    Lines3[14].X := 195.736; Lines3[14].Z := 249.746; Lines3[14].F := 800; Lines3[14].CMD := 1; Lines3[14].Param := 0; // G1 Linear [Op5 P1]
    Lines3[15].X := 194.386; Lines3[15].Z := 250.431; Lines3[15].F := 800; Lines3[15].CMD := 1; Lines3[15].Param := 0; // G1 Linear [Op5 P1]
    Lines3[16].X := 193.033; Lines3[16].Z := 251.111; Lines3[16].F := 800; Lines3[16].CMD := 1; Lines3[16].Param := 0; // G1 Linear [Op5 P1]
    Lines3[17].X := 191.451; Lines3[17].Z := 251.899; Lines3[17].F := 800; Lines3[17].CMD := 1; Lines3[17].Param := 0; // G1 Linear [Op5 P1]
    Lines3[18].X := 192.808; Lines3[18].Z := 251.224; Lines3[18].F := 800; Lines3[18].CMD := 1; Lines3[18].Param := 0; // G1 Linear [Op5 P1]
    Lines3[19].X := 194.161; Lines3[19].Z := 250.545; Lines3[19].F := 800; Lines3[19].CMD := 1; Lines3[19].Param := 0; // G1 Linear [Op5 P1]
    Lines3[20].X := 195.736; Lines3[20].Z := 249.746; Lines3[20].F := 800; Lines3[20].CMD := 1; Lines3[20].Param := 0; // G1 Linear [Op5 P1]
    Lines3[21].X := 197.082; Lines3[21].Z := 249.056; Lines3[21].F := 800; Lines3[21].CMD := 1; Lines3[21].Param := 0; // G1 Linear [Op5 P1]
    Lines3[22].X := 198.426; Lines3[22].Z := 248.363; Lines3[22].F := 800; Lines3[22].CMD := 1; Lines3[22].Param := 0; // G1 Linear [Op5 P1]
    Lines3[23].X := 199.990; Lines3[23].Z := 247.547; Lines3[23].F := 800; Lines3[23].CMD := 1; Lines3[23].Param := 0; // G1 Linear [Op5 P1]
    Lines3[24].X := 201.328; Lines3[24].Z := 246.844; Lines3[24].F := 800; Lines3[24].CMD := 1; Lines3[24].Param := 0; // G1 Linear [Op5 P1]
    Lines3[25].X := 202.662; Lines3[25].Z := 246.135; Lines3[25].F := 800; Lines3[25].CMD := 1; Lines3[25].Param := 0; // G1 Linear [Op5 P1]
    Lines3[26].X := 203.994; Lines3[26].Z := 245.422; Lines3[26].F := 800; Lines3[26].CMD := 1; Lines3[26].Param := 0; // G1 Linear [Op5 P1]
    Lines3[27].X := 205.322; Lines3[27].Z := 244.705; Lines3[27].F := 800; Lines3[27].CMD := 1; Lines3[27].Param := 0; // G1 Linear [Op5 P1]
    Lines3[28].X := 206.648; Lines3[28].Z := 243.983; Lines3[28].F := 800; Lines3[28].CMD := 1; Lines3[28].Param := 0; // G1 Linear [Op5 P1]
    Lines3[29].X := 208.190; Lines3[29].Z := 243.136; Lines3[29].F := 800; Lines3[29].CMD := 1; Lines3[29].Param := 0; // G1 Linear [Op5 P1]
    Lines3[30].X := 209.510; Lines3[30].Z := 242.404; Lines3[30].F := 800; Lines3[30].CMD := 1; Lines3[30].Param := 0; // G1 Linear [Op5 P1]
    Lines3[31].X := 210.826; Lines3[31].Z := 241.668; Lines3[31].F := 800; Lines3[31].CMD := 1; Lines3[31].Param := 0; // G1 Linear [Op5 P1]
    Lines3[32].X := 212.139; Lines3[32].Z := 240.927; Lines3[32].F := 800; Lines3[32].CMD := 1; Lines3[32].Param := 0; // G1 Linear [Op5 P1]
    Lines3[33].X := 213.667; Lines3[33].Z := 240.057; Lines3[33].F := 800; Lines3[33].CMD := 1; Lines3[33].Param := 0; // G1 Linear [Op5 P1]
    Lines3[34].X := 214.974; Lines3[34].Z := 239.307; Lines3[34].F := 800; Lines3[34].CMD := 1; Lines3[34].Param := 0; // G1 Linear [Op5 P1]
    Lines3[35].X := 216.278; Lines3[35].Z := 238.552; Lines3[35].F := 800; Lines3[35].CMD := 1; Lines3[35].Param := 0; // G1 Linear [Op5 P1]
    Lines3[36].X := 217.796; Lines3[36].Z := 237.666; Lines3[36].F := 800; Lines3[36].CMD := 1; Lines3[36].Param := 0; // G1 Linear [Op5 P1]
    Lines3[37].X := 219.093; Lines3[37].Z := 236.901; Lines3[37].F := 800; Lines3[37].CMD := 1; Lines3[37].Param := 0; // G1 Linear [Op5 P1]
    Lines3[38].X := 220.603; Lines3[38].Z := 236.003; Lines3[38].F := 800; Lines3[38].CMD := 1; Lines3[38].Param := 0; // G1 Linear [Op5 P1]
    Lines3[39].X := 221.894; Lines3[39].Z := 235.228; Lines3[39].F := 800; Lines3[39].CMD := 1; Lines3[39].Param := 0; // G1 Linear [Op5 P1]
    Lines3[40].X := 223.182; Lines3[40].Z := 234.449; Lines3[40].F := 800; Lines3[40].CMD := 1; Lines3[40].Param := 0; // G1 Linear [Op5 P1]
    Lines3[41].X := 224.467; Lines3[41].Z := 233.666; Lines3[41].F := 800; Lines3[41].CMD := 1; Lines3[41].Param := 0; // G1 Linear [Op5 P1]
    Lines3[42].X := 225.750; Lines3[42].Z := 232.878; Lines3[42].F := 800; Lines3[42].CMD := 1; Lines3[42].Param := 0; // G1 Linear [Op5 P1]
    Lines3[43].X := 227.029; Lines3[43].Z := 232.085; Lines3[43].F := 800; Lines3[43].CMD := 1; Lines3[43].Param := 0; // G1 Linear [Op5 P1]
    Lines3[44].X := 228.518; Lines3[44].Z := 231.155; Lines3[44].F := 800; Lines3[44].CMD := 1; Lines3[44].Param := 0; // G1 Linear [Op5 P1]
    Lines3[45].X := 229.791; Lines3[45].Z := 230.352; Lines3[45].F := 800; Lines3[45].CMD := 1; Lines3[45].Param := 0; // G1 Linear [Op5 P1]
    Lines3[46].X := 231.060; Lines3[46].Z := 229.545; Lines3[46].F := 800; Lines3[46].CMD := 1; Lines3[46].Param := 0; // G1 Linear [Op5 P1]
    Lines3[47].X := 232.327; Lines3[47].Z := 228.734; Lines3[47].F := 800; Lines3[47].CMD := 1; Lines3[47].Param := 0; // G1 Linear [Op5 P1]
    Lines3[48].X := 233.802; Lines3[48].Z := 227.782; Lines3[48].F := 800; Lines3[48].CMD := 1; Lines3[48].Param := 0; // G1 Linear [Op5 P1]
    Lines3[49].X := 235.062; Lines3[49].Z := 226.960; Lines3[49].F := 800; Lines3[49].CMD := 1; Lines3[49].Param := 0; // G1 Linear [Op5 P1]
    Lines3[50].X := 236.320; Lines3[50].Z := 226.135; Lines3[50].F := 800; Lines3[50].CMD := 1; Lines3[50].Param := 0; // G1 Linear [Op5 P1]
    Lines3[51].X := 237.783; Lines3[51].Z := 225.165; Lines3[51].F := 800; Lines3[51].CMD := 1; Lines3[51].Param := 0; // G1 Linear [Op5 P1]
    Lines3[52].X := 239.034; Lines3[52].Z := 224.330; Lines3[52].F := 800; Lines3[52].CMD := 1; Lines3[52].Param := 0; // G1 Linear [Op5 P1]
    Lines3[53].X := 240.283; Lines3[53].Z := 223.490; Lines3[53].F := 800; Lines3[53].CMD := 1; Lines3[53].Param := 0; // G1 Linear [Op5 P1]
    Lines3[54].X := 241.528; Lines3[54].Z := 222.645; Lines3[54].F := 800; Lines3[54].CMD := 1; Lines3[54].Param := 0; // G1 Linear [Op5 P1]
    Lines3[55].X := 242.977; Lines3[55].Z := 221.654; Lines3[55].F := 800; Lines3[55].CMD := 1; Lines3[55].Param := 0; // G1 Linear [Op5 P1]
    Lines3[56].X := 244.216; Lines3[56].Z := 220.800; Lines3[56].F := 800; Lines3[56].CMD := 1; Lines3[56].Param := 0; // G1 Linear [Op5 P1]
    Lines3[57].X := 245.452; Lines3[57].Z := 219.941; Lines3[57].F := 800; Lines3[57].CMD := 1; Lines3[57].Param := 0; // G1 Linear [Op5 P1]
    Lines3[58].X := 246.685; Lines3[58].Z := 219.078; Lines3[58].F := 800; Lines3[58].CMD := 1; Lines3[58].Param := 0; // G1 Linear [Op5 P1]
    Lines3[59].X := 248.119; Lines3[59].Z := 218.065; Lines3[59].F := 800; Lines3[59].CMD := 1; Lines3[59].Param := 0; // G1 Linear [Op5 P1]
    Lines3[60].X := 249.346; Lines3[60].Z := 217.191; Lines3[60].F := 800; Lines3[60].CMD := 1; Lines3[60].Param := 0; // G1 Linear [Op5 P1]
    Lines3[61].X := 250.570; Lines3[61].Z := 216.314; Lines3[61].F := 800; Lines3[61].CMD := 1; Lines3[61].Param := 0; // G1 Linear [Op5 P1]
    Lines3[62].X := 251.790; Lines3[62].Z := 215.431; Lines3[62].F := 800; Lines3[62].CMD := 1; Lines3[62].Param := 0; // G1 Linear [Op5 P1]
    Lines3[63].X := 253.211; Lines3[63].Z := 214.396; Lines3[63].F := 800; Lines3[63].CMD := 1; Lines3[63].Param := 0; // G1 Linear [Op5 P1]
    Lines3[64].X := 254.425; Lines3[64].Z := 213.504; Lines3[64].F := 800; Lines3[64].CMD := 1; Lines3[64].Param := 0; // G1 Linear [Op5 P1]
    Lines3[65].X := 255.636; Lines3[65].Z := 212.608; Lines3[65].F := 800; Lines3[65].CMD := 1; Lines3[65].Param := 0; // G1 Linear [Op5 P1]
    Lines3[66].X := 256.844; Lines3[66].Z := 211.707; Lines3[66].F := 800; Lines3[66].CMD := 1; Lines3[66].Param := 0; // G1 Linear [Op5 P1]
    Lines3[67].X := 258.050; Lines3[67].Z := 210.801; Lines3[67].F := 800; Lines3[67].CMD := 1; Lines3[67].Param := 0; // G1 Linear [Op5 P1]
    Lines3[68].X := 259.252; Lines3[68].Z := 209.891; Lines3[68].F := 800; Lines3[68].CMD := 1; Lines3[68].Param := 0; // G1 Linear [Op5 P1]
    Lines3[69].X := 260.651; Lines3[69].Z := 208.824; Lines3[69].F := 800; Lines3[69].CMD := 1; Lines3[69].Param := 0; // G1 Linear [Op5 P1]
    Lines3[70].X := 261.847; Lines3[70].Z := 207.904; Lines3[70].F := 800; Lines3[70].CMD := 1; Lines3[70].Param := 0; // G1 Linear [Op5 P1]
    Lines3[71].X := 263.239; Lines3[71].Z := 206.825; Lines3[71].F := 800; Lines3[71].CMD := 1; Lines3[71].Param := 0; // G1 Linear [Op5 P1]
    Lines3[72].X := 264.428; Lines3[72].Z := 205.895; Lines3[72].F := 800; Lines3[72].CMD := 1; Lines3[72].Param := 0; // G1 Linear [Op5 P1]
    Lines3[73].X := 265.615; Lines3[73].Z := 204.961; Lines3[73].F := 800; Lines3[73].CMD := 1; Lines3[73].Param := 0; // G1 Linear [Op5 P1]
    Lines3[74].X := 266.799; Lines3[74].Z := 204.022; Lines3[74].F := 800; Lines3[74].CMD := 1; Lines3[74].Param := 0; // G1 Linear [Op5 P1]
    Lines3[75].X := 267.980; Lines3[75].Z := 203.079; Lines3[75].F := 800; Lines3[75].CMD := 1; Lines3[75].Param := 0; // G1 Linear [Op5 P1]
    Lines3[76].X := 269.353; Lines3[76].Z := 201.973; Lines3[76].F := 800; Lines3[76].CMD := 1; Lines3[76].Param := 0; // G1 Linear [Op5 P1]
    Lines3[77].X := 270.528; Lines3[77].Z := 201.020; Lines3[77].F := 800; Lines3[77].CMD := 1; Lines3[77].Param := 0; // G1 Linear [Op5 P1]
    Lines3[78].X := 271.699; Lines3[78].Z := 200.062; Lines3[78].F := 800; Lines3[78].CMD := 1; Lines3[78].Param := 0; // G1 Linear [Op5 P1]
    Lines3[79].X := 273.062; Lines3[79].Z := 198.939; Lines3[79].F := 800; Lines3[79].CMD := 1; Lines3[79].Param := 0; // G1 Linear [Op5 P1]
    Lines3[80].X := 274.227; Lines3[80].Z := 197.972; Lines3[80].F := 800; Lines3[80].CMD := 1; Lines3[80].Param := 0; // G1 Linear [Op5 P1]
    Lines3[81].X := 275.389; Lines3[81].Z := 197.000; Lines3[81].F := 800; Lines3[81].CMD := 1; Lines3[81].Param := 0; // G1 Linear [Op5 P1]
    Lines3[82].X := 265.389; Lines3[82].Z := 187.000; Lines3[82].F := 0; Lines3[82].CMD := 0; Lines3[82].Param := 0; // G0 Rapid [Op5 P1]
    Lines3[83].X := 265.389; Lines3[83].Z := 187.000; Lines3[83].F := 0; Lines3[83].CMD := 20; Lines3[83].Param := 80; // Spindle ON 800 RPM [Op5 P1]
    Lines3[84].X := 275.449; Lines3[84].Z := 181.000; Lines3[84].F := 0; Lines3[84].CMD := 0; Lines3[84].Param := 0; // G0 Rapid [Op6 P1]
    Lines3[85].X := 275.382; Lines3[85].Z := 201.000; Lines3[85].F := 500; Lines3[85].CMD := 1; Lines3[85].Param := 0; // G1 Linear [Op6 P1]
    Lines3[86].X := 274.126; Lines3[86].Z := 202.242; Lines3[86].F := 500; Lines3[86].CMD := 1; Lines3[86].Param := 0; // G1 Linear [Op6 P1]
    Lines3[87].X := 273.046; Lines3[87].Z := 203.302; Lines3[87].F := 500; Lines3[87].CMD := 1; Lines3[87].Param := 0; // G1 Linear [Op6 P1]
    Lines3[88].X := 271.782; Lines3[88].Z := 204.534; Lines3[88].F := 500; Lines3[88].CMD := 1; Lines3[88].Param := 0; // G1 Linear [Op6 P1]
    Lines3[89].X := 270.695; Lines3[89].Z := 205.586; Lines3[89].F := 500; Lines3[89].CMD := 1; Lines3[89].Param := 0; // G1 Linear [Op6 P1]
    Lines3[90].X := 269.605; Lines3[90].Z := 206.633; Lines3[90].F := 500; Lines3[90].CMD := 1; Lines3[90].Param := 0; // G1 Linear [Op6 P1]
    Lines3[91].X := 268.329; Lines3[91].Z := 207.851; Lines3[91].F := 500; Lines3[91].CMD := 1; Lines3[91].Param := 0; // G1 Linear [Op6 P1]
    Lines3[92].X := 267.050; Lines3[92].Z := 209.063; Lines3[92].F := 500; Lines3[92].CMD := 1; Lines3[92].Param := 0; // G1 Linear [Op6 P1]
    Lines3[93].X := 265.949; Lines3[93].Z := 210.097; Lines3[93].F := 500; Lines3[93].CMD := 1; Lines3[93].Param := 0; // G1 Linear [Op6 P1]
    Lines3[94].X := 264.662; Lines3[94].Z := 211.300; Lines3[94].F := 500; Lines3[94].CMD := 1; Lines3[94].Param := 0; // G1 Linear [Op6 P1]
    Lines3[95].X := 263.555; Lines3[95].Z := 212.326; Lines3[95].F := 500; Lines3[95].CMD := 1; Lines3[95].Param := 0; // G1 Linear [Op6 P1]
    Lines3[96].X := 262.259; Lines3[96].Z := 213.518; Lines3[96].F := 500; Lines3[96].CMD := 1; Lines3[96].Param := 0; // G1 Linear [Op6 P1]
    Lines3[97].X := 261.145; Lines3[97].Z := 214.535; Lines3[97].F := 500; Lines3[97].CMD := 1; Lines3[97].Param := 0; // G1 Linear [Op6 P1]
    Lines3[98].X := 259.842; Lines3[98].Z := 215.717; Lines3[98].F := 500; Lines3[98].CMD := 1; Lines3[98].Param := 0; // G1 Linear [Op6 P1]
    Lines3[99].X := 258.722; Lines3[99].Z := 216.726; Lines3[99].F := 500; Lines3[99].CMD := 1; Lines3[99].Param := 0; // G1 Linear [Op6 P1]
    Lines4[0].X := 257.598; Lines4[0].Z := 217.731; Lines4[0].F := 500; Lines4[0].CMD := 1; Lines4[0].Param := 0; // G1 Linear [Op6 P1]
    Lines4[1].X := 256.283; Lines4[1].Z := 218.899; Lines4[1].F := 500; Lines4[1].CMD := 1; Lines4[1].Param := 0; // G1 Linear [Op6 P1]
    Lines4[2].X := 255.153; Lines4[2].Z := 219.895; Lines4[2].F := 500; Lines4[2].CMD := 1; Lines4[2].Param := 0; // G1 Linear [Op6 P1]
    Lines4[3].X := 253.831; Lines4[3].Z := 221.053; Lines4[3].F := 500; Lines4[3].CMD := 1; Lines4[3].Param := 0; // G1 Linear [Op6 P1]
    Lines4[4].X := 252.694; Lines4[4].Z := 222.041; Lines4[4].F := 500; Lines4[4].CMD := 1; Lines4[4].Param := 0; // G1 Linear [Op6 P1]
    Lines4[5].X := 251.363; Lines4[5].Z := 223.189; Lines4[5].F := 500; Lines4[5].CMD := 1; Lines4[5].Param := 0; // G1 Linear [Op6 P1]
    Lines4[6].X := 250.219; Lines4[6].Z := 224.168; Lines4[6].F := 500; Lines4[6].CMD := 1; Lines4[6].Param := 0; // G1 Linear [Op6 P1]
    Lines4[7].X := 248.881; Lines4[7].Z := 225.306; Lines4[7].F := 500; Lines4[7].CMD := 1; Lines4[7].Param := 0; // G1 Linear [Op6 P1]
    Lines4[8].X := 247.539; Lines4[8].Z := 226.438; Lines4[8].F := 500; Lines4[8].CMD := 1; Lines4[8].Param := 0; // G1 Linear [Op6 P1]
    Lines4[9].X := 246.384; Lines4[9].Z := 227.404; Lines4[9].F := 500; Lines4[9].CMD := 1; Lines4[9].Param := 0; // G1 Linear [Op6 P1]
    Lines4[10].X := 245.227; Lines4[10].Z := 228.366; Lines4[10].F := 500; Lines4[10].CMD := 1; Lines4[10].Param := 0; // G1 Linear [Op6 P1]
    Lines4[11].X := 243.873; Lines4[11].Z := 229.484; Lines4[11].F := 500; Lines4[11].CMD := 1; Lines4[11].Param := 0; // G1 Linear [Op6 P1]
    Lines4[12].X := 242.709; Lines4[12].Z := 230.438; Lines4[12].F := 500; Lines4[12].CMD := 1; Lines4[12].Param := 0; // G1 Linear [Op6 P1]
    Lines4[13].X := 241.348; Lines4[13].Z := 231.546; Lines4[13].F := 500; Lines4[13].CMD := 1; Lines4[13].Param := 0; // G1 Linear [Op6 P1]
    Lines4[14].X := 240.177; Lines4[14].Z := 232.491; Lines4[14].F := 500; Lines4[14].CMD := 1; Lines4[14].Param := 0; // G1 Linear [Op6 P1]
    Lines4[15].X := 238.807; Lines4[15].Z := 233.589; Lines4[15].F := 500; Lines4[15].CMD := 1; Lines4[15].Param := 0; // G1 Linear [Op6 P1]
    Lines4[16].X := 237.630; Lines4[16].Z := 234.526; Lines4[16].F := 500; Lines4[16].CMD := 1; Lines4[16].Param := 0; // G1 Linear [Op6 P1]
    Lines4[17].X := 236.253; Lines4[17].Z := 235.613; Lines4[17].F := 500; Lines4[17].CMD := 1; Lines4[17].Param := 0; // G1 Linear [Op6 P1]
    Lines4[18].X := 234.871; Lines4[18].Z := 236.696; Lines4[18].F := 500; Lines4[18].CMD := 1; Lines4[18].Param := 0; // G1 Linear [Op6 P1]
    Lines4[19].X := 233.683; Lines4[19].Z := 237.619; Lines4[19].F := 500; Lines4[19].CMD := 1; Lines4[19].Param := 0; // G1 Linear [Op6 P1]
    Lines4[20].X := 232.492; Lines4[20].Z := 238.539; Lines4[20].F := 500; Lines4[20].CMD := 1; Lines4[20].Param := 0; // G1 Linear [Op6 P1]
    Lines4[21].X := 231.099; Lines4[21].Z := 239.607; Lines4[21].F := 500; Lines4[21].CMD := 1; Lines4[21].Param := 0; // G1 Linear [Op6 P1]
    Lines4[22].X := 229.902; Lines4[22].Z := 240.518; Lines4[22].F := 500; Lines4[22].CMD := 1; Lines4[22].Param := 0; // G1 Linear [Op6 P1]
    Lines4[23].X := 228.501; Lines4[23].Z := 241.576; Lines4[23].F := 500; Lines4[23].CMD := 1; Lines4[23].Param := 0; // G1 Linear [Op6 P1]
    Lines4[24].X := 227.296; Lines4[24].Z := 242.478; Lines4[24].F := 500; Lines4[24].CMD := 1; Lines4[24].Param := 0; // G1 Linear [Op6 P1]
    Lines4[25].X := 225.888; Lines4[25].Z := 243.526; Lines4[25].F := 500; Lines4[25].CMD := 1; Lines4[25].Param := 0; // G1 Linear [Op6 P1]
    Lines4[26].X := 224.677; Lines4[26].Z := 244.420; Lines4[26].F := 500; Lines4[26].CMD := 1; Lines4[26].Param := 0; // G1 Linear [Op6 P1]
    Lines4[27].X := 223.260; Lines4[27].Z := 245.458; Lines4[27].F := 500; Lines4[27].CMD := 1; Lines4[27].Param := 0; // G1 Linear [Op6 P1]
    Lines4[28].X := 222.042; Lines4[28].Z := 246.344; Lines4[28].F := 500; Lines4[28].CMD := 1; Lines4[28].Param := 0; // G1 Linear [Op6 P1]
    Lines4[29].X := 220.618; Lines4[29].Z := 247.372; Lines4[29].F := 500; Lines4[29].CMD := 1; Lines4[29].Param := 0; // G1 Linear [Op6 P1]
    Lines4[30].X := 218.166; Lines4[30].Z := 249.122; Lines4[30].F := 500; Lines4[30].CMD := 1; Lines4[30].Param := 0; // G1 Linear [Op6 P1]
    Lines4[31].X := 216.935; Lines4[31].Z := 249.991; Lines4[31].F := 500; Lines4[31].CMD := 1; Lines4[31].Param := 0; // G1 Linear [Op6 P1]
    Lines4[32].X := 215.496; Lines4[32].Z := 251.000; Lines4[32].F := 500; Lines4[32].CMD := 1; Lines4[32].Param := 0; // G1 Linear [Op6 P1]
    Lines4[33].X := 214.258; Lines4[33].Z := 251.860; Lines4[33].F := 500; Lines4[33].CMD := 1; Lines4[33].Param := 0; // G1 Linear [Op6 P1]
    Lines4[34].X := 212.811; Lines4[34].Z := 252.859; Lines4[34].F := 500; Lines4[34].CMD := 1; Lines4[34].Param := 0; // G1 Linear [Op6 P1]
    Lines4[35].X := 211.567; Lines4[35].Z := 253.711; Lines4[35].F := 500; Lines4[35].CMD := 1; Lines4[35].Param := 0; // G1 Linear [Op6 P1]
    Lines4[36].X := 210.111; Lines4[36].Z := 254.700; Lines4[36].F := 500; Lines4[36].CMD := 1; Lines4[36].Param := 0; // G1 Linear [Op6 P1]
    Lines4[37].X := 208.861; Lines4[37].Z := 255.543; Lines4[37].F := 500; Lines4[37].CMD := 1; Lines4[37].Param := 0; // G1 Linear [Op6 P1]
    Lines4[38].X := 207.397; Lines4[38].Z := 256.522; Lines4[38].F := 500; Lines4[38].CMD := 1; Lines4[38].Param := 0; // G1 Linear [Op6 P1]
    Lines4[39].X := 206.140; Lines4[39].Z := 257.357; Lines4[39].F := 500; Lines4[39].CMD := 1; Lines4[39].Param := 0; // G1 Linear [Op6 P1]
    Lines4[40].X := 204.669; Lines4[40].Z := 258.326; Lines4[40].F := 500; Lines4[40].CMD := 1; Lines4[40].Param := 0; // G1 Linear [Op6 P1]
    Lines4[41].X := 203.405; Lines4[41].Z := 259.153; Lines4[41].F := 500; Lines4[41].CMD := 1; Lines4[41].Param := 0; // G1 Linear [Op6 P1]
    Lines4[42].X := 201.926; Lines4[42].Z := 260.112; Lines4[42].F := 500; Lines4[42].CMD := 1; Lines4[42].Param := 0; // G1 Linear [Op6 P1]
    Lines4[43].X := 200.655; Lines4[43].Z := 260.929; Lines4[43].F := 500; Lines4[43].CMD := 1; Lines4[43].Param := 0; // G1 Linear [Op6 P1]
    Lines4[44].X := 199.168; Lines4[44].Z := 261.878; Lines4[44].F := 500; Lines4[44].CMD := 1; Lines4[44].Param := 0; // G1 Linear [Op6 P1]
    Lines4[45].X := 197.891; Lines4[45].Z := 262.688; Lines4[45].F := 500; Lines4[45].CMD := 1; Lines4[45].Param := 0; // G1 Linear [Op6 P1]
    Lines4[46].X := 196.396; Lines4[46].Z := 263.627; Lines4[46].F := 500; Lines4[46].CMD := 1; Lines4[46].Param := 0; // G1 Linear [Op6 P1]
    Lines4[47].X := 195.112; Lines4[47].Z := 264.428; Lines4[47].F := 500; Lines4[47].CMD := 1; Lines4[47].Param := 0; // G1 Linear [Op6 P1]
    Lines4[48].X := 193.609; Lines4[48].Z := 265.357; Lines4[48].F := 500; Lines4[48].CMD := 1; Lines4[48].Param := 0; // G1 Linear [Op6 P1]
    Lines4[49].X := 183.609; Lines4[49].Z := 255.357; Lines4[49].F := 0; Lines4[49].CMD := 0; Lines4[49].Param := 0; // G0 Rapid [Op6 P1]
    Lines4[50].X := 183.609; Lines4[50].Z := 255.357; Lines4[50].F := 0; Lines4[50].CMD := 20; Lines4[50].Param := 80; // Spindle ON 800 RPM [Op6 P1]
    Lines4[51].X := 275.849; Lines4[51].Z := 181.000; Lines4[51].F := 0; Lines4[51].CMD := 0; Lines4[51].Param := 0; // G0 Rapid [Op7 P1]
    Lines4[52].X := 275.769; Lines4[52].Z := 205.000; Lines4[52].F := 500; Lines4[52].CMD := 1; Lines4[52].Param := 0; // G1 Linear [Op7 P1]
    Lines4[53].X := 274.621; Lines4[53].Z := 206.345; Lines4[53].F := 500; Lines4[53].CMD := 1; Lines4[53].Param := 0; // G1 Linear [Op7 P1]
    Lines4[54].X := 273.634; Lines4[54].Z := 207.493; Lines4[54].F := 500; Lines4[54].CMD := 1; Lines4[54].Param := 0; // G1 Linear [Op7 P1]
    Lines4[55].X := 272.478; Lines4[55].Z := 208.829; Lines4[55].F := 500; Lines4[55].CMD := 1; Lines4[55].Param := 0; // G1 Linear [Op7 P1]
    Lines4[56].X := 271.483; Lines4[56].Z := 209.969; Lines4[56].F := 500; Lines4[56].CMD := 1; Lines4[56].Param := 0; // G1 Linear [Op7 P1]
    Lines4[57].X := 270.319; Lines4[57].Z := 211.295; Lines4[57].F := 500; Lines4[57].CMD := 1; Lines4[57].Param := 0; // G1 Linear [Op7 P1]
    Lines4[58].X := 269.317; Lines4[58].Z := 212.428; Lines4[58].F := 500; Lines4[58].CMD := 1; Lines4[58].Param := 0; // G1 Linear [Op7 P1]
    Lines4[59].X := 268.143; Lines4[59].Z := 213.745; Lines4[59].F := 500; Lines4[59].CMD := 1; Lines4[59].Param := 0; // G1 Linear [Op7 P1]
    Lines4[60].X := 267.134; Lines4[60].Z := 214.870; Lines4[60].F := 500; Lines4[60].CMD := 1; Lines4[60].Param := 0; // G1 Linear [Op7 P1]
    Lines4[61].X := 265.952; Lines4[61].Z := 216.178; Lines4[61].F := 500; Lines4[61].CMD := 1; Lines4[61].Param := 0; // G1 Linear [Op7 P1]
    Lines4[62].X := 264.935; Lines4[62].Z := 217.295; Lines4[62].F := 500; Lines4[62].CMD := 1; Lines4[62].Param := 0; // G1 Linear [Op7 P1]
    Lines4[63].X := 263.915; Lines4[63].Z := 218.408; Lines4[63].F := 500; Lines4[63].CMD := 1; Lines4[63].Param := 0; // G1 Linear [Op7 P1]
    Lines4[64].X := 262.720; Lines4[64].Z := 219.702; Lines4[64].F := 500; Lines4[64].CMD := 1; Lines4[64].Param := 0; // G1 Linear [Op7 P1]
    Lines4[65].X := 261.521; Lines4[65].Z := 220.992; Lines4[65].F := 500; Lines4[65].CMD := 1; Lines4[65].Param := 0; // G1 Linear [Op7 P1]
    Lines4[66].X := 260.490; Lines4[66].Z := 222.093; Lines4[66].F := 500; Lines4[66].CMD := 1; Lines4[66].Param := 0; // G1 Linear [Op7 P1]
    Lines4[67].X := 259.282; Lines4[67].Z := 223.373; Lines4[67].F := 500; Lines4[67].CMD := 1; Lines4[67].Param := 0; // G1 Linear [Op7 P1]
    Lines4[68].X := 258.243; Lines4[68].Z := 224.466; Lines4[68].F := 500; Lines4[68].CMD := 1; Lines4[68].Param := 0; // G1 Linear [Op7 P1]
    Lines4[69].X := 257.026; Lines4[69].Z := 225.737; Lines4[69].F := 500; Lines4[69].CMD := 1; Lines4[69].Param := 0; // G1 Linear [Op7 P1]
    Lines4[70].X := 255.980; Lines4[70].Z := 226.823; Lines4[70].F := 500; Lines4[70].CMD := 1; Lines4[70].Param := 0; // G1 Linear [Op7 P1]
    Lines4[71].X := 254.755; Lines4[71].Z := 228.084; Lines4[71].F := 500; Lines4[71].CMD := 1; Lines4[71].Param := 0; // G1 Linear [Op7 P1]
    Lines4[72].X := 253.701; Lines4[72].Z := 229.162; Lines4[72].F := 500; Lines4[72].CMD := 1; Lines4[72].Param := 0; // G1 Linear [Op7 P1]
    Lines4[73].X := 252.644; Lines4[73].Z := 230.236; Lines4[73].F := 500; Lines4[73].CMD := 1; Lines4[73].Param := 0; // G1 Linear [Op7 P1]
    Lines4[74].X := 251.407; Lines4[74].Z := 231.484; Lines4[74].F := 500; Lines4[74].CMD := 1; Lines4[74].Param := 0; // G1 Linear [Op7 P1]
    Lines4[75].X := 250.164; Lines4[75].Z := 232.727; Lines4[75].F := 500; Lines4[75].CMD := 1; Lines4[75].Param := 0; // G1 Linear [Op7 P1]
    Lines4[76].X := 249.096; Lines4[76].Z := 233.789; Lines4[76].F := 500; Lines4[76].CMD := 1; Lines4[76].Param := 0; // G1 Linear [Op7 P1]
    Lines4[77].X := 248.024; Lines4[77].Z := 234.847; Lines4[77].F := 500; Lines4[77].CMD := 1; Lines4[77].Param := 0; // G1 Linear [Op7 P1]
    Lines4[78].X := 246.769; Lines4[78].Z := 236.076; Lines4[78].F := 500; Lines4[78].CMD := 1; Lines4[78].Param := 0; // G1 Linear [Op7 P1]
    Lines4[79].X := 245.509; Lines4[79].Z := 237.301; Lines4[79].F := 500; Lines4[79].CMD := 1; Lines4[79].Param := 0; // G1 Linear [Op7 P1]
    Lines4[80].X := 244.426; Lines4[80].Z := 238.347; Lines4[80].F := 500; Lines4[80].CMD := 1; Lines4[80].Param := 0; // G1 Linear [Op7 P1]
    Lines4[81].X := 243.339; Lines4[81].Z := 239.389; Lines4[81].F := 500; Lines4[81].CMD := 1; Lines4[81].Param := 0; // G1 Linear [Op7 P1]
    Lines4[82].X := 242.067; Lines4[82].Z := 240.601; Lines4[82].F := 500; Lines4[82].CMD := 1; Lines4[82].Param := 0; // G1 Linear [Op7 P1]
    Lines4[83].X := 240.973; Lines4[83].Z := 241.635; Lines4[83].F := 500; Lines4[83].CMD := 1; Lines4[83].Param := 0; // G1 Linear [Op7 P1]
    Lines4[84].X := 239.692; Lines4[84].Z := 242.837; Lines4[84].F := 500; Lines4[84].CMD := 1; Lines4[84].Param := 0; // G1 Linear [Op7 P1]
    Lines4[85].X := 238.591; Lines4[85].Z := 243.863; Lines4[85].F := 500; Lines4[85].CMD := 1; Lines4[85].Param := 0; // G1 Linear [Op7 P1]
    Lines4[86].X := 237.302; Lines4[86].Z := 245.056; Lines4[86].F := 500; Lines4[86].CMD := 1; Lines4[86].Param := 0; // G1 Linear [Op7 P1]
    Lines4[87].X := 236.193; Lines4[87].Z := 246.075; Lines4[87].F := 500; Lines4[87].CMD := 1; Lines4[87].Param := 0; // G1 Linear [Op7 P1]
    Lines4[88].X := 234.895; Lines4[88].Z := 247.258; Lines4[88].F := 500; Lines4[88].CMD := 1; Lines4[88].Param := 0; // G1 Linear [Op7 P1]
    Lines4[89].X := 233.779; Lines4[89].Z := 248.269; Lines4[89].F := 500; Lines4[89].CMD := 1; Lines4[89].Param := 0; // G1 Linear [Op7 P1]
    Lines4[90].X := 232.472; Lines4[90].Z := 249.443; Lines4[90].F := 500; Lines4[90].CMD := 1; Lines4[90].Param := 0; // G1 Linear [Op7 P1]
    Lines4[91].X := 231.348; Lines4[91].Z := 250.446; Lines4[91].F := 500; Lines4[91].CMD := 1; Lines4[91].Param := 0; // G1 Linear [Op7 P1]
    Lines4[92].X := 230.033; Lines4[92].Z := 251.611; Lines4[92].F := 500; Lines4[92].CMD := 1; Lines4[92].Param := 0; // G1 Linear [Op7 P1]
    Lines4[93].X := 228.713; Lines4[93].Z := 252.772; Lines4[93].F := 500; Lines4[93].CMD := 1; Lines4[93].Param := 0; // G1 Linear [Op7 P1]
    Lines4[94].X := 227.578; Lines4[94].Z := 253.762; Lines4[94].F := 500; Lines4[94].CMD := 1; Lines4[94].Param := 0; // G1 Linear [Op7 P1]
    Lines4[95].X := 226.250; Lines4[95].Z := 254.913; Lines4[95].F := 500; Lines4[95].CMD := 1; Lines4[95].Param := 0; // G1 Linear [Op7 P1]
    Lines4[96].X := 225.107; Lines4[96].Z := 255.896; Lines4[96].F := 500; Lines4[96].CMD := 1; Lines4[96].Param := 0; // G1 Linear [Op7 P1]
    Lines4[97].X := 223.962; Lines4[97].Z := 256.875; Lines4[97].F := 500; Lines4[97].CMD := 1; Lines4[97].Param := 0; // G1 Linear [Op7 P1]
    Lines4[98].X := 222.621; Lines4[98].Z := 258.012; Lines4[98].F := 500; Lines4[98].CMD := 1; Lines4[98].Param := 0; // G1 Linear [Op7 P1]
    Lines4[99].X := 221.467; Lines4[99].Z := 258.984; Lines4[99].F := 500; Lines4[99].CMD := 1; Lines4[99].Param := 0; // G1 Linear [Op7 P1]
    Lines5[0].X := 220.118; Lines5[0].Z := 260.112; Lines5[0].F := 500; Lines5[0].CMD := 1; Lines5[0].Param := 0; // G1 Linear [Op7 P1]
    Lines5[1].X := 218.957; Lines5[1].Z := 261.075; Lines5[1].F := 500; Lines5[1].CMD := 1; Lines5[1].Param := 0; // G1 Linear [Op7 P1]
    Lines5[2].X := 217.599; Lines5[2].Z := 262.194; Lines5[2].F := 500; Lines5[2].CMD := 1; Lines5[2].Param := 0; // G1 Linear [Op7 P1]
    Lines5[3].X := 216.236; Lines5[3].Z := 263.308; Lines5[3].F := 500; Lines5[3].CMD := 1; Lines5[3].Param := 0; // G1 Linear [Op7 P1]
    Lines5[4].X := 215.064; Lines5[4].Z := 264.259; Lines5[4].F := 500; Lines5[4].CMD := 1; Lines5[4].Param := 0; // G1 Linear [Op7 P1]
    Lines5[5].X := 213.889; Lines5[5].Z := 265.207; Lines5[5].F := 500; Lines5[5].CMD := 1; Lines5[5].Param := 0; // G1 Linear [Op7 P1]
    Lines5[6].X := 212.513; Lines5[6].Z := 266.307; Lines5[6].F := 500; Lines5[6].CMD := 1; Lines5[6].Param := 0; // G1 Linear [Op7 P1]
    Lines5[7].X := 211.330; Lines5[7].Z := 267.247; Lines5[7].F := 500; Lines5[7].CMD := 1; Lines5[7].Param := 0; // G1 Linear [Op7 P1]
    Lines5[8].X := 209.946; Lines5[8].Z := 268.338; Lines5[8].F := 500; Lines5[8].CMD := 1; Lines5[8].Param := 0; // G1 Linear [Op7 P1]
    Lines5[9].X := 208.756; Lines5[9].Z := 269.270; Lines5[9].F := 500; Lines5[9].CMD := 1; Lines5[9].Param := 0; // G1 Linear [Op7 P1]
    Lines5[10].X := 207.363; Lines5[10].Z := 270.352; Lines5[10].F := 500; Lines5[10].CMD := 1; Lines5[10].Param := 0; // G1 Linear [Op7 P1]
    Lines5[11].X := 206.166; Lines5[11].Z := 271.276; Lines5[11].F := 500; Lines5[11].CMD := 1; Lines5[11].Param := 0; // G1 Linear [Op7 P1]
    Lines5[12].X := 204.764; Lines5[12].Z := 272.349; Lines5[12].F := 500; Lines5[12].CMD := 1; Lines5[12].Param := 0; // G1 Linear [Op7 P1]
    Lines5[13].X := 203.559; Lines5[13].Z := 273.265; Lines5[13].F := 500; Lines5[13].CMD := 1; Lines5[13].Param := 0; // G1 Linear [Op7 P1]
    Lines5[14].X := 202.149; Lines5[14].Z := 274.329; Lines5[14].F := 500; Lines5[14].CMD := 1; Lines5[14].Param := 0; // G1 Linear [Op7 P1]
    Lines5[15].X := 200.937; Lines5[15].Z := 275.236; Lines5[15].F := 500; Lines5[15].CMD := 1; Lines5[15].Param := 0; // G1 Linear [Op7 P1]
    Lines5[16].X := 199.518; Lines5[16].Z := 276.291; Lines5[16].F := 500; Lines5[16].CMD := 1; Lines5[16].Param := 0; // G1 Linear [Op7 P1]
    Lines5[17].X := 189.518; Lines5[17].Z := 266.291; Lines5[17].F := 0; Lines5[17].CMD := 0; Lines5[17].Param := 0; // G0 Rapid [Op7 P1]
    Lines5[18].X := 189.518; Lines5[18].Z := 266.291; Lines5[18].F := 0; Lines5[18].CMD := 20; Lines5[18].Param := 80; // Spindle ON 800 RPM [Op7 P1]
    Lines5[19].X := 275.832; Lines5[19].Z := 186.000; Lines5[19].F := 0; Lines5[19].CMD := 0; Lines5[19].Param := 0; // G0 Rapid [Op8 P1]
    Lines5[20].X := 275.759; Lines5[20].Z := 208.000; Lines5[20].F := 800; Lines5[20].CMD := 1; Lines5[20].Param := 0; // G1 Linear [Op8 P1]
    Lines5[21].X := 274.834; Lines5[21].Z := 209.198; Lines5[21].F := 800; Lines5[21].CMD := 1; Lines5[21].Param := 0; // G1 Linear [Op8 P1]
    Lines5[22].X := 273.751; Lines5[22].Z := 210.591; Lines5[22].F := 800; Lines5[22].CMD := 1; Lines5[22].Param := 0; // G1 Linear [Op8 P1]
    Lines5[23].X := 272.663; Lines5[23].Z := 211.980; Lines5[23].F := 800; Lines5[23].CMD := 1; Lines5[23].Param := 0; // G1 Linear [Op8 P1]
    Lines5[24].X := 271.570; Lines5[24].Z := 213.365; Lines5[24].F := 800; Lines5[24].CMD := 1; Lines5[24].Param := 0; // G1 Linear [Op8 P1]
    Lines5[25].X := 270.473; Lines5[25].Z := 214.745; Lines5[25].F := 800; Lines5[25].CMD := 1; Lines5[25].Param := 0; // G1 Linear [Op8 P1]
    Lines5[26].X := 269.372; Lines5[26].Z := 216.121; Lines5[26].F := 800; Lines5[26].CMD := 1; Lines5[26].Param := 0; // G1 Linear [Op8 P1]
    Lines5[27].X := 268.424; Lines5[27].Z := 217.296; Lines5[27].F := 800; Lines5[27].CMD := 1; Lines5[27].Param := 0; // G1 Linear [Op8 P1]
    Lines5[28].X := 267.314; Lines5[28].Z := 218.664; Lines5[28].F := 800; Lines5[28].CMD := 1; Lines5[28].Param := 0; // G1 Linear [Op8 P1]
    Lines5[29].X := 266.199; Lines5[29].Z := 220.027; Lines5[29].F := 800; Lines5[29].CMD := 1; Lines5[29].Param := 0; // G1 Linear [Op8 P1]
    Lines5[30].X := 265.080; Lines5[30].Z := 221.386; Lines5[30].F := 800; Lines5[30].CMD := 1; Lines5[30].Param := 0; // G1 Linear [Op8 P1]
    Lines5[31].X := 264.117; Lines5[31].Z := 222.547; Lines5[31].F := 800; Lines5[31].CMD := 1; Lines5[31].Param := 0; // G1 Linear [Op8 P1]
    Lines5[32].X := 262.990; Lines5[32].Z := 223.898; Lines5[32].F := 800; Lines5[32].CMD := 1; Lines5[32].Param := 0; // G1 Linear [Op8 P1]
    Lines5[33].X := 261.858; Lines5[33].Z := 225.244; Lines5[33].F := 800; Lines5[33].CMD := 1; Lines5[33].Param := 0; // G1 Linear [Op8 P1]
    Lines5[34].X := 260.721; Lines5[34].Z := 226.586; Lines5[34].F := 800; Lines5[34].CMD := 1; Lines5[34].Param := 0; // G1 Linear [Op8 P1]
    Lines5[35].X := 259.580; Lines5[35].Z := 227.924; Lines5[35].F := 800; Lines5[35].CMD := 1; Lines5[35].Param := 0; // G1 Linear [Op8 P1]
    Lines5[36].X := 258.598; Lines5[36].Z := 229.067; Lines5[36].F := 800; Lines5[36].CMD := 1; Lines5[36].Param := 0; // G1 Linear [Op8 P1]
    Lines5[37].X := 257.613; Lines5[37].Z := 230.206; Lines5[37].F := 800; Lines5[37].CMD := 1; Lines5[37].Param := 0; // G1 Linear [Op8 P1]
    Lines5[38].X := 256.459; Lines5[38].Z := 231.532; Lines5[38].F := 800; Lines5[38].CMD := 1; Lines5[38].Param := 0; // G1 Linear [Op8 P1]
    Lines5[39].X := 255.301; Lines5[39].Z := 232.853; Lines5[39].F := 800; Lines5[39].CMD := 1; Lines5[39].Param := 0; // G1 Linear [Op8 P1]
    Lines5[40].X := 254.138; Lines5[40].Z := 234.170; Lines5[40].F := 800; Lines5[40].CMD := 1; Lines5[40].Param := 0; // G1 Linear [Op8 P1]
    Lines5[41].X := 253.138; Lines5[41].Z := 235.295; Lines5[41].F := 800; Lines5[41].CMD := 1; Lines5[41].Param := 0; // G1 Linear [Op8 P1]
    Lines5[42].X := 251.966; Lines5[42].Z := 236.604; Lines5[42].F := 800; Lines5[42].CMD := 1; Lines5[42].Param := 0; // G1 Linear [Op8 P1]
    Lines5[43].X := 250.791; Lines5[43].Z := 237.908; Lines5[43].F := 800; Lines5[43].CMD := 1; Lines5[43].Param := 0; // G1 Linear [Op8 P1]
    Lines5[44].X := 249.610; Lines5[44].Z := 239.208; Lines5[44].F := 800; Lines5[44].CMD := 1; Lines5[44].Param := 0; // G1 Linear [Op8 P1]
    Lines5[45].X := 248.595; Lines5[45].Z := 240.319; Lines5[45].F := 800; Lines5[45].CMD := 1; Lines5[45].Param := 0; // G1 Linear [Op8 P1]
    Lines5[46].X := 247.406; Lines5[46].Z := 241.610; Lines5[46].F := 800; Lines5[46].CMD := 1; Lines5[46].Param := 0; // G1 Linear [Op8 P1]
    Lines5[47].X := 246.213; Lines5[47].Z := 242.898; Lines5[47].F := 800; Lines5[47].CMD := 1; Lines5[47].Param := 0; // G1 Linear [Op8 P1]
    Lines5[48].X := 245.015; Lines5[48].Z := 244.181; Lines5[48].F := 800; Lines5[48].CMD := 1; Lines5[48].Param := 0; // G1 Linear [Op8 P1]
    Lines5[49].X := 243.812; Lines5[49].Z := 245.459; Lines5[49].F := 800; Lines5[49].CMD := 1; Lines5[49].Param := 0; // G1 Linear [Op8 P1]
    Lines5[50].X := 242.605; Lines5[50].Z := 246.733; Lines5[50].F := 800; Lines5[50].CMD := 1; Lines5[50].Param := 0; // G1 Linear [Op8 P1]
    Lines5[51].X := 241.567; Lines5[51].Z := 247.822; Lines5[51].F := 800; Lines5[51].CMD := 1; Lines5[51].Param := 0; // G1 Linear [Op8 P1]
    Lines5[52].X := 240.351; Lines5[52].Z := 249.088; Lines5[52].F := 800; Lines5[52].CMD := 1; Lines5[52].Param := 0; // G1 Linear [Op8 P1]
    Lines5[53].X := 239.306; Lines5[53].Z := 250.170; Lines5[53].F := 800; Lines5[53].CMD := 1; Lines5[53].Param := 0; // G1 Linear [Op8 P1]
    Lines5[54].X := 238.082; Lines5[54].Z := 251.427; Lines5[54].F := 800; Lines5[54].CMD := 1; Lines5[54].Param := 0; // G1 Linear [Op8 P1]
    Lines5[55].X := 237.029; Lines5[55].Z := 252.502; Lines5[55].F := 800; Lines5[55].CMD := 1; Lines5[55].Param := 0; // G1 Linear [Op8 P1]
    Lines5[56].X := 235.797; Lines5[56].Z := 253.752; Lines5[56].F := 800; Lines5[56].CMD := 1; Lines5[56].Param := 0; // G1 Linear [Op8 P1]
    Lines5[57].X := 234.560; Lines5[57].Z := 254.997; Lines5[57].F := 800; Lines5[57].CMD := 1; Lines5[57].Param := 0; // G1 Linear [Op8 P1]
    Lines5[58].X := 233.318; Lines5[58].Z := 256.238; Lines5[58].F := 800; Lines5[58].CMD := 1; Lines5[58].Param := 0; // G1 Linear [Op8 P1]
    Lines5[59].X := 232.250; Lines5[59].Z := 257.298; Lines5[59].F := 800; Lines5[59].CMD := 1; Lines5[59].Param := 0; // G1 Linear [Op8 P1]
    Lines5[60].X := 231.000; Lines5[60].Z := 258.531; Lines5[60].F := 800; Lines5[60].CMD := 1; Lines5[60].Param := 0; // G1 Linear [Op8 P1]
    Lines5[61].X := 229.745; Lines5[61].Z := 259.759; Lines5[61].F := 800; Lines5[61].CMD := 1; Lines5[61].Param := 0; // G1 Linear [Op8 P1]
    Lines5[62].X := 228.486; Lines5[62].Z := 260.983; Lines5[62].F := 800; Lines5[62].CMD := 1; Lines5[62].Param := 0; // G1 Linear [Op8 P1]
    Lines5[63].X := 227.403; Lines5[63].Z := 262.029; Lines5[63].F := 800; Lines5[63].CMD := 1; Lines5[63].Param := 0; // G1 Linear [Op8 P1]
    Lines5[64].X := 226.136; Lines5[64].Z := 263.245; Lines5[64].F := 800; Lines5[64].CMD := 1; Lines5[64].Param := 0; // G1 Linear [Op8 P1]
    Lines5[65].X := 225.045; Lines5[65].Z := 264.283; Lines5[65].F := 800; Lines5[65].CMD := 1; Lines5[65].Param := 0; // G1 Linear [Op8 P1]
    Lines5[66].X := 223.769; Lines5[66].Z := 265.491; Lines5[66].F := 800; Lines5[66].CMD := 1; Lines5[66].Param := 0; // G1 Linear [Op8 P1]
    Lines5[67].X := 222.489; Lines5[67].Z := 266.694; Lines5[67].F := 800; Lines5[67].CMD := 1; Lines5[67].Param := 0; // G1 Linear [Op8 P1]
    Lines5[68].X := 221.203; Lines5[68].Z := 267.893; Lines5[68].F := 800; Lines5[68].CMD := 1; Lines5[68].Param := 0; // G1 Linear [Op8 P1]
    Lines5[69].X := 220.098; Lines5[69].Z := 268.917; Lines5[69].F := 800; Lines5[69].CMD := 1; Lines5[69].Param := 0; // G1 Linear [Op8 P1]
    Lines5[70].X := 218.804; Lines5[70].Z := 270.108; Lines5[70].F := 800; Lines5[70].CMD := 1; Lines5[70].Param := 0; // G1 Linear [Op8 P1]
    Lines5[71].X := 217.506; Lines5[71].Z := 271.294; Lines5[71].F := 800; Lines5[71].CMD := 1; Lines5[71].Param := 0; // G1 Linear [Op8 P1]
    Lines5[72].X := 216.203; Lines5[72].Z := 272.476; Lines5[72].F := 800; Lines5[72].CMD := 1; Lines5[72].Param := 0; // G1 Linear [Op8 P1]
    Lines5[73].X := 215.083; Lines5[73].Z := 273.486; Lines5[73].F := 800; Lines5[73].CMD := 1; Lines5[73].Param := 0; // G1 Linear [Op8 P1]
    Lines5[74].X := 213.772; Lines5[74].Z := 274.659; Lines5[74].F := 800; Lines5[74].CMD := 1; Lines5[74].Param := 0; // G1 Linear [Op8 P1]
    Lines5[75].X := 212.456; Lines5[75].Z := 275.829; Lines5[75].F := 800; Lines5[75].CMD := 1; Lines5[75].Param := 0; // G1 Linear [Op8 P1]
    Lines5[76].X := 211.135; Lines5[76].Z := 276.994; Lines5[76].F := 800; Lines5[76].CMD := 1; Lines5[76].Param := 0; // G1 Linear [Op8 P1]
    Lines5[77].X := 209.811; Lines5[77].Z := 278.154; Lines5[77].F := 800; Lines5[77].CMD := 1; Lines5[77].Param := 0; // G1 Linear [Op8 P1]
    Lines5[78].X := 208.671; Lines5[78].Z := 279.146; Lines5[78].F := 800; Lines5[78].CMD := 1; Lines5[78].Param := 0; // G1 Linear [Op8 P1]
    Lines5[79].X := 207.338; Lines5[79].Z := 280.298; Lines5[79].F := 800; Lines5[79].CMD := 1; Lines5[79].Param := 0; // G1 Linear [Op8 P1]
    Lines5[80].X := 206.000; Lines5[80].Z := 281.446; Lines5[80].F := 800; Lines5[80].CMD := 1; Lines5[80].Param := 0; // G1 Linear [Op8 P1]
    Lines5[81].X := 204.849; Lines5[81].Z := 282.427; Lines5[81].F := 800; Lines5[81].CMD := 1; Lines5[81].Param := 0; // G1 Linear [Op8 P1]
    Lines5[82].X := 203.503; Lines5[82].Z := 283.567; Lines5[82].F := 800; Lines5[82].CMD := 1; Lines5[82].Param := 0; // G1 Linear [Op8 P1]
    Lines5[83].X := 202.152; Lines5[83].Z := 284.702; Lines5[83].F := 800; Lines5[83].CMD := 1; Lines5[83].Param := 0; // G1 Linear [Op8 P1]
    Lines5[84].X := 200.796; Lines5[84].Z := 285.833; Lines5[84].F := 800; Lines5[84].CMD := 1; Lines5[84].Param := 0; // G1 Linear [Op8 P1]
    Lines5[85].X := 190.796; Lines5[85].Z := 275.833; Lines5[85].F := 0; Lines5[85].CMD := 0; Lines5[85].Param := 0; // G0 Rapid [Op8 P1]
    Lines5[86].X := 190.796; Lines5[86].Z := 275.833; Lines5[86].F := 0; Lines5[86].CMD := 20; Lines5[86].Param := 80; // Spindle ON 800 RPM [Op8 P1]
    Lines5[87].X := 190.796; Lines5[87].Z := 275.833; Lines5[87].F := 0; Lines5[87].CMD := 41; Lines5[87].Param := 2; // M41 (Clamp On) P2 [Op9 P1]
    Lines5[88].X := 275.769; Lines5[88].Z := 205.000; Lines5[88].F := 0; Lines5[88].CMD := 0; Lines5[88].Param := 0; // G0 Rapid [Op9 P1]
    Lines5[89].X := 275.745; Lines5[89].Z := 212.000; Lines5[89].F := 800; Lines5[89].CMD := 1; Lines5[89].Param := 0; // G1 Linear [Op9 P1]
    Lines5[90].X := 274.770; Lines5[90].Z := 213.474; Lines5[90].F := 800; Lines5[90].CMD := 1; Lines5[90].Param := 0; // G1 Linear [Op9 P1]
    Lines5[91].X := 273.790; Lines5[91].Z := 214.943; Lines5[91].F := 800; Lines5[91].CMD := 1; Lines5[91].Param := 0; // G1 Linear [Op9 P1]
    Lines5[92].X := 272.945; Lines5[92].Z := 216.199; Lines5[92].F := 800; Lines5[92].CMD := 1; Lines5[92].Param := 0; // G1 Linear [Op9 P1]
    Lines5[93].X := 271.955; Lines5[93].Z := 217.661; Lines5[93].F := 800; Lines5[93].CMD := 1; Lines5[93].Param := 0; // G1 Linear [Op9 P1]
    Lines5[94].X := 271.102; Lines5[94].Z := 218.910; Lines5[94].F := 800; Lines5[94].CMD := 1; Lines5[94].Param := 0; // G1 Linear [Op9 P1]
    Lines5[95].X := 270.102; Lines5[95].Z := 220.363; Lines5[95].F := 800; Lines5[95].CMD := 1; Lines5[95].Param := 0; // G1 Linear [Op9 P1]
    Lines5[96].X := 269.241; Lines5[96].Z := 221.606; Lines5[96].F := 800; Lines5[96].CMD := 1; Lines5[96].Param := 0; // G1 Linear [Op9 P1]
    Lines5[97].X := 268.232; Lines5[97].Z := 223.051; Lines5[97].F := 800; Lines5[97].CMD := 1; Lines5[97].Param := 0; // G1 Linear [Op9 P1]
    Lines5[98].X := 267.363; Lines5[98].Z := 224.287; Lines5[98].F := 800; Lines5[98].CMD := 1; Lines5[98].Param := 0; // G1 Linear [Op9 P1]
    Lines5[99].X := 266.344; Lines5[99].Z := 225.724; Lines5[99].F := 800; Lines5[99].CMD := 1; Lines5[99].Param := 0; // G1 Linear [Op9 P1]
    Lines6[0].X := 265.467; Lines6[0].Z := 226.953; Lines6[0].F := 800; Lines6[0].CMD := 1; Lines6[0].Param := 0; // G1 Linear [Op9 P1]
    Lines6[1].X := 264.438; Lines6[1].Z := 228.382; Lines6[1].F := 800; Lines6[1].CMD := 1; Lines6[1].Param := 0; // G1 Linear [Op9 P1]
    Lines6[2].X := 263.553; Lines6[2].Z := 229.604; Lines6[2].F := 800; Lines6[2].CMD := 1; Lines6[2].Param := 0; // G1 Linear [Op9 P1]
    Lines6[3].X := 262.514; Lines6[3].Z := 231.025; Lines6[3].F := 800; Lines6[3].CMD := 1; Lines6[3].Param := 0; // G1 Linear [Op9 P1]
    Lines6[4].X := 261.621; Lines6[4].Z := 232.240; Lines6[4].F := 800; Lines6[4].CMD := 1; Lines6[4].Param := 0; // G1 Linear [Op9 P1]
    Lines6[5].X := 260.573; Lines6[5].Z := 233.653; Lines6[5].F := 800; Lines6[5].CMD := 1; Lines6[5].Param := 0; // G1 Linear [Op9 P1]
    Lines6[6].X := 259.671; Lines6[6].Z := 234.861; Lines6[6].F := 800; Lines6[6].CMD := 1; Lines6[6].Param := 0; // G1 Linear [Op9 P1]
    Lines6[7].X := 258.614; Lines6[7].Z := 236.267; Lines6[7].F := 800; Lines6[7].CMD := 1; Lines6[7].Param := 0; // G1 Linear [Op9 P1]
    Lines6[8].X := 257.703; Lines6[8].Z := 237.468; Lines6[8].F := 800; Lines6[8].CMD := 1; Lines6[8].Param := 0; // G1 Linear [Op9 P1]
    Lines6[9].X := 256.637; Lines6[9].Z := 238.865; Lines6[9].F := 800; Lines6[9].CMD := 1; Lines6[9].Param := 0; // G1 Linear [Op9 P1]
    Lines6[10].X := 255.718; Lines6[10].Z := 240.059; Lines6[10].F := 800; Lines6[10].CMD := 1; Lines6[10].Param := 0; // G1 Linear [Op9 P1]
    Lines6[11].X := 254.642; Lines6[11].Z := 241.448; Lines6[11].F := 800; Lines6[11].CMD := 1; Lines6[11].Param := 0; // G1 Linear [Op9 P1]
    Lines6[12].X := 253.715; Lines6[12].Z := 242.636; Lines6[12].F := 800; Lines6[12].CMD := 1; Lines6[12].Param := 0; // G1 Linear [Op9 P1]
    Lines6[13].X := 252.629; Lines6[13].Z := 244.017; Lines6[13].F := 800; Lines6[13].CMD := 1; Lines6[13].Param := 0; // G1 Linear [Op9 P1]
    Lines6[14].X := 251.538; Lines6[14].Z := 245.394; Lines6[14].F := 800; Lines6[14].CMD := 1; Lines6[14].Param := 0; // G1 Linear [Op9 P1]
    Lines6[15].X := 250.598; Lines6[15].Z := 246.571; Lines6[15].F := 800; Lines6[15].CMD := 1; Lines6[15].Param := 0; // G1 Linear [Op9 P1]
    Lines6[16].X := 249.655; Lines6[16].Z := 247.744; Lines6[16].F := 800; Lines6[16].CMD := 1; Lines6[16].Param := 0; // G1 Linear [Op9 P1]
    Lines6[17].X := 248.550; Lines6[17].Z := 249.109; Lines6[17].F := 800; Lines6[17].CMD := 1; Lines6[17].Param := 0; // G1 Linear [Op9 P1]
    Lines6[18].X := 247.599; Lines6[18].Z := 250.276; Lines6[18].F := 800; Lines6[18].CMD := 1; Lines6[18].Param := 0; // G1 Linear [Op9 P1]
    Lines6[19].X := 246.484; Lines6[19].Z := 251.633; Lines6[19].F := 800; Lines6[19].CMD := 1; Lines6[19].Param := 0; // G1 Linear [Op9 P1]
    Lines6[20].X := 245.364; Lines6[20].Z := 252.986; Lines6[20].F := 800; Lines6[20].CMD := 1; Lines6[20].Param := 0; // G1 Linear [Op9 P1]
    Lines6[21].X := 244.400; Lines6[21].Z := 254.142; Lines6[21].F := 800; Lines6[21].CMD := 1; Lines6[21].Param := 0; // G1 Linear [Op9 P1]
    Lines6[22].X := 243.432; Lines6[22].Z := 255.295; Lines6[22].F := 800; Lines6[22].CMD := 1; Lines6[22].Param := 0; // G1 Linear [Op9 P1]
    Lines6[23].X := 242.298; Lines6[23].Z := 256.636; Lines6[23].F := 800; Lines6[23].CMD := 1; Lines6[23].Param := 0; // G1 Linear [Op9 P1]
    Lines6[24].X := 241.159; Lines6[24].Z := 257.973; Lines6[24].F := 800; Lines6[24].CMD := 1; Lines6[24].Param := 0; // G1 Linear [Op9 P1]
    Lines6[25].X := 240.015; Lines6[25].Z := 259.306; Lines6[25].F := 800; Lines6[25].CMD := 1; Lines6[25].Param := 0; // G1 Linear [Op9 P1]
    Lines6[26].X := 238.866; Lines6[26].Z := 260.634; Lines6[26].F := 800; Lines6[26].CMD := 1; Lines6[26].Param := 0; // G1 Linear [Op9 P1]
    Lines6[27].X := 237.876; Lines6[27].Z := 261.769; Lines6[27].F := 800; Lines6[27].CMD := 1; Lines6[27].Param := 0; // G1 Linear [Op9 P1]
    Lines6[28].X := 236.883; Lines6[28].Z := 262.901; Lines6[28].F := 800; Lines6[28].CMD := 1; Lines6[28].Param := 0; // G1 Linear [Op9 P1]
    Lines6[29].X := 235.720; Lines6[29].Z := 264.217; Lines6[29].F := 800; Lines6[29].CMD := 1; Lines6[29].Param := 0; // G1 Linear [Op9 P1]
    Lines6[30].X := 234.718; Lines6[30].Z := 265.342; Lines6[30].F := 800; Lines6[30].CMD := 1; Lines6[30].Param := 0; // G1 Linear [Op9 P1]
    Lines6[31].X := 233.545; Lines6[31].Z := 266.651; Lines6[31].F := 800; Lines6[31].CMD := 1; Lines6[31].Param := 0; // G1 Linear [Op9 P1]
    Lines6[32].X := 232.536; Lines6[32].Z := 267.769; Lines6[32].F := 800; Lines6[32].CMD := 1; Lines6[32].Param := 0; // G1 Linear [Op9 P1]
    Lines6[33].X := 231.353; Lines6[33].Z := 269.069; Lines6[33].F := 800; Lines6[33].CMD := 1; Lines6[33].Param := 0; // G1 Linear [Op9 P1]
    Lines6[34].X := 230.336; Lines6[34].Z := 270.180; Lines6[34].F := 800; Lines6[34].CMD := 1; Lines6[34].Param := 0; // G1 Linear [Op9 P1]
    Lines6[35].X := 229.143; Lines6[35].Z := 271.473; Lines6[35].F := 800; Lines6[35].CMD := 1; Lines6[35].Param := 0; // G1 Linear [Op9 P1]
    Lines6[36].X := 228.117; Lines6[36].Z := 272.577; Lines6[36].F := 800; Lines6[36].CMD := 1; Lines6[36].Param := 0; // G1 Linear [Op9 P1]
    Lines6[37].X := 226.916; Lines6[37].Z := 273.861; Lines6[37].F := 800; Lines6[37].CMD := 1; Lines6[37].Param := 0; // G1 Linear [Op9 P1]
    Lines6[38].X := 225.881; Lines6[38].Z := 274.959; Lines6[38].F := 800; Lines6[38].CMD := 1; Lines6[38].Param := 0; // G1 Linear [Op9 P1]
    Lines6[39].X := 224.670; Lines6[39].Z := 276.235; Lines6[39].F := 800; Lines6[39].CMD := 1; Lines6[39].Param := 0; // G1 Linear [Op9 P1]
    Lines6[40].X := 223.628; Lines6[40].Z := 277.326; Lines6[40].F := 800; Lines6[40].CMD := 1; Lines6[40].Param := 0; // G1 Linear [Op9 P1]
    Lines6[41].X := 222.407; Lines6[41].Z := 278.594; Lines6[41].F := 800; Lines6[41].CMD := 1; Lines6[41].Param := 0; // G1 Linear [Op9 P1]
    Lines6[42].X := 221.356; Lines6[42].Z := 279.678; Lines6[42].F := 800; Lines6[42].CMD := 1; Lines6[42].Param := 0; // G1 Linear [Op9 P1]
    Lines6[43].X := 220.126; Lines6[43].Z := 280.938; Lines6[43].F := 800; Lines6[43].CMD := 1; Lines6[43].Param := 0; // G1 Linear [Op9 P1]
    Lines6[44].X := 218.890; Lines6[44].Z := 282.194; Lines6[44].F := 800; Lines6[44].CMD := 1; Lines6[44].Param := 0; // G1 Linear [Op9 P1]
    Lines6[45].X := 217.827; Lines6[45].Z := 283.267; Lines6[45].F := 800; Lines6[45].CMD := 1; Lines6[45].Param := 0; // G1 Linear [Op9 P1]
    Lines6[46].X := 216.760; Lines6[46].Z := 284.337; Lines6[46].F := 800; Lines6[46].CMD := 1; Lines6[46].Param := 0; // G1 Linear [Op9 P1]
    Lines6[47].X := 215.510; Lines6[47].Z := 285.581; Lines6[47].F := 800; Lines6[47].CMD := 1; Lines6[47].Param := 0; // G1 Linear [Op9 P1]
    Lines6[48].X := 214.435; Lines6[48].Z := 286.644; Lines6[48].F := 800; Lines6[48].CMD := 1; Lines6[48].Param := 0; // G1 Linear [Op9 P1]
    Lines6[49].X := 213.175; Lines6[49].Z := 287.881; Lines6[49].F := 800; Lines6[49].CMD := 1; Lines6[49].Param := 0; // G1 Linear [Op9 P1]
    Lines6[50].X := 212.092; Lines6[50].Z := 288.937; Lines6[50].F := 800; Lines6[50].CMD := 1; Lines6[50].Param := 0; // G1 Linear [Op9 P1]
    Lines6[51].X := 210.823; Lines6[51].Z := 290.165; Lines6[51].F := 800; Lines6[51].CMD := 1; Lines6[51].Param := 0; // G1 Linear [Op9 P1]
    Lines6[52].X := 209.549; Lines6[52].Z := 291.389; Lines6[52].F := 800; Lines6[52].CMD := 1; Lines6[52].Param := 0; // G1 Linear [Op9 P1]
    Lines6[53].X := 208.453; Lines6[53].Z := 292.435; Lines6[53].F := 800; Lines6[53].CMD := 1; Lines6[53].Param := 0; // G1 Linear [Op9 P1]
    Lines6[54].X := 198.453; Lines6[54].Z := 282.435; Lines6[54].F := 0; Lines6[54].CMD := 0; Lines6[54].Param := 0; // G0 Rapid [Op9 P1]
    Lines6[55].X := 198.453; Lines6[55].Z := 282.435; Lines6[55].F := 0; Lines6[55].CMD := 20; Lines6[55].Param := 80; // Spindle ON 800 RPM [Op9 P1]
    Lines6[56].X := 275.938; Lines6[56].Z := 184.077; Lines6[56].F := 0; Lines6[56].CMD := 0; Lines6[56].Param := 0; // G0 Rapid [Op10 P1]
    Lines6[57].X := 275.832; Lines6[57].Z := 216.077; Lines6[57].F := 800; Lines6[57].CMD := 1; Lines6[57].Param := 0; // G1 Linear [Op10 P1]
    Lines6[58].X := 274.933; Lines6[58].Z := 217.600; Lines6[58].F := 800; Lines6[58].CMD := 1; Lines6[58].Param := 0; // G1 Linear [Op10 P1]
    Lines6[59].X := 274.159; Lines6[59].Z := 218.902; Lines6[59].F := 800; Lines6[59].CMD := 1; Lines6[59].Param := 0; // G1 Linear [Op10 P1]
    Lines6[60].X := 273.250; Lines6[60].Z := 220.418; Lines6[60].F := 800; Lines6[60].CMD := 1; Lines6[60].Param := 0; // G1 Linear [Op10 P1]
    Lines6[61].X := 272.467; Lines6[61].Z := 221.714; Lines6[61].F := 800; Lines6[61].CMD := 1; Lines6[61].Param := 0; // G1 Linear [Op10 P1]
    Lines6[62].X := 271.548; Lines6[62].Z := 223.222; Lines6[62].F := 800; Lines6[62].CMD := 1; Lines6[62].Param := 0; // G1 Linear [Op10 P1]
    Lines6[63].X := 270.624; Lines6[63].Z := 224.726; Lines6[63].F := 800; Lines6[63].CMD := 1; Lines6[63].Param := 0; // G1 Linear [Op10 P1]
    Lines6[64].X := 269.828; Lines6[64].Z := 226.012; Lines6[64].F := 800; Lines6[64].CMD := 1; Lines6[64].Param := 0; // G1 Linear [Op10 P1]
    Lines6[65].X := 268.894; Lines6[65].Z := 227.508; Lines6[65].F := 800; Lines6[65].CMD := 1; Lines6[65].Param := 0; // G1 Linear [Op10 P1]
    Lines6[66].X := 268.089; Lines6[66].Z := 228.788; Lines6[66].F := 800; Lines6[66].CMD := 1; Lines6[66].Param := 0; // G1 Linear [Op10 P1]
    Lines6[67].X := 267.145; Lines6[67].Z := 230.277; Lines6[67].F := 800; Lines6[67].CMD := 1; Lines6[67].Param := 0; // G1 Linear [Op10 P1]
    Lines6[68].X := 266.332; Lines6[68].Z := 231.550; Lines6[68].F := 800; Lines6[68].CMD := 1; Lines6[68].Param := 0; // G1 Linear [Op10 P1]
    Lines6[69].X := 265.378; Lines6[69].Z := 233.031; Lines6[69].F := 800; Lines6[69].CMD := 1; Lines6[69].Param := 0; // G1 Linear [Op10 P1]
    Lines6[70].X := 264.556; Lines6[70].Z := 234.298; Lines6[70].F := 800; Lines6[70].CMD := 1; Lines6[70].Param := 0; // G1 Linear [Op10 P1]
    Lines6[71].X := 263.592; Lines6[71].Z := 235.772; Lines6[71].F := 800; Lines6[71].CMD := 1; Lines6[71].Param := 0; // G1 Linear [Op10 P1]
    Lines6[72].X := 262.761; Lines6[72].Z := 237.032; Lines6[72].F := 800; Lines6[72].CMD := 1; Lines6[72].Param := 0; // G1 Linear [Op10 P1]
    Lines6[73].X := 261.787; Lines6[73].Z := 238.498; Lines6[73].F := 800; Lines6[73].CMD := 1; Lines6[73].Param := 0; // G1 Linear [Op10 P1]
    Lines6[74].X := 260.948; Lines6[74].Z := 239.752; Lines6[74].F := 800; Lines6[74].CMD := 1; Lines6[74].Param := 0; // G1 Linear [Op10 P1]
    Lines6[75].X := 259.964; Lines6[75].Z := 241.211; Lines6[75].F := 800; Lines6[75].CMD := 1; Lines6[75].Param := 0; // G1 Linear [Op10 P1]
    Lines6[76].X := 259.117; Lines6[76].Z := 242.458; Lines6[76].F := 800; Lines6[76].CMD := 1; Lines6[76].Param := 0; // G1 Linear [Op10 P1]
    Lines6[77].X := 258.123; Lines6[77].Z := 243.910; Lines6[77].F := 800; Lines6[77].CMD := 1; Lines6[77].Param := 0; // G1 Linear [Op10 P1]
    Lines6[78].X := 257.267; Lines6[78].Z := 245.151; Lines6[78].F := 800; Lines6[78].CMD := 1; Lines6[78].Param := 0; // G1 Linear [Op10 P1]
    Lines6[79].X := 256.263; Lines6[79].Z := 246.595; Lines6[79].F := 800; Lines6[79].CMD := 1; Lines6[79].Param := 0; // G1 Linear [Op10 P1]
    Lines6[80].X := 255.253; Lines6[80].Z := 248.034; Lines6[80].F := 800; Lines6[80].CMD := 1; Lines6[80].Param := 0; // G1 Linear [Op10 P1]
    Lines6[81].X := 254.384; Lines6[81].Z := 249.265; Lines6[81].F := 800; Lines6[81].CMD := 1; Lines6[81].Param := 0; // G1 Linear [Op10 P1]
    Lines6[82].X := 253.365; Lines6[82].Z := 250.698; Lines6[82].F := 800; Lines6[82].CMD := 1; Lines6[82].Param := 0; // G1 Linear [Op10 P1]
    Lines6[83].X := 252.487; Lines6[83].Z := 251.922; Lines6[83].F := 800; Lines6[83].CMD := 1; Lines6[83].Param := 0; // G1 Linear [Op10 P1]
    Lines6[84].X := 251.458; Lines6[84].Z := 253.347; Lines6[84].F := 800; Lines6[84].CMD := 1; Lines6[84].Param := 0; // G1 Linear [Op10 P1]
    Lines6[85].X := 250.571; Lines6[85].Z := 254.565; Lines6[85].F := 800; Lines6[85].CMD := 1; Lines6[85].Param := 0; // G1 Linear [Op10 P1]
    Lines6[86].X := 249.532; Lines6[86].Z := 255.982; Lines6[86].F := 800; Lines6[86].CMD := 1; Lines6[86].Param := 0; // G1 Linear [Op10 P1]
    Lines6[87].X := 248.637; Lines6[87].Z := 257.194; Lines6[87].F := 800; Lines6[87].CMD := 1; Lines6[87].Param := 0; // G1 Linear [Op10 P1]
    Lines6[88].X := 247.738; Lines6[88].Z := 258.403; Lines6[88].F := 800; Lines6[88].CMD := 1; Lines6[88].Param := 0; // G1 Linear [Op10 P1]
    Lines6[89].X := 246.684; Lines6[89].Z := 259.809; Lines6[89].F := 800; Lines6[89].CMD := 1; Lines6[89].Param := 0; // G1 Linear [Op10 P1]
    Lines6[90].X := 245.776; Lines6[90].Z := 261.011; Lines6[90].F := 800; Lines6[90].CMD := 1; Lines6[90].Param := 0; // G1 Linear [Op10 P1]
    Lines6[91].X := 244.712; Lines6[91].Z := 262.410; Lines6[91].F := 800; Lines6[91].CMD := 1; Lines6[91].Param := 0; // G1 Linear [Op10 P1]
    Lines6[92].X := 243.796; Lines6[92].Z := 263.606; Lines6[92].F := 800; Lines6[92].CMD := 1; Lines6[92].Param := 0; // G1 Linear [Op10 P1]
    Lines6[93].X := 242.722; Lines6[93].Z := 264.997; Lines6[93].F := 800; Lines6[93].CMD := 1; Lines6[93].Param := 0; // G1 Linear [Op10 P1]
    Lines6[94].X := 241.798; Lines6[94].Z := 266.186; Lines6[94].F := 800; Lines6[94].CMD := 1; Lines6[94].Param := 0; // G1 Linear [Op10 P1]
    Lines6[95].X := 240.714; Lines6[95].Z := 267.570; Lines6[95].F := 800; Lines6[95].CMD := 1; Lines6[95].Param := 0; // G1 Linear [Op10 P1]
    Lines6[96].X := 239.625; Lines6[96].Z := 268.950; Lines6[96].F := 800; Lines6[96].CMD := 1; Lines6[96].Param := 0; // G1 Linear [Op10 P1]
    Lines6[97].X := 238.687; Lines6[97].Z := 270.129; Lines6[97].F := 800; Lines6[97].CMD := 1; Lines6[97].Param := 0; // G1 Linear [Op10 P1]
    Lines6[98].X := 237.745; Lines6[98].Z := 271.306; Lines6[98].F := 800; Lines6[98].CMD := 1; Lines6[98].Param := 0; // G1 Linear [Op10 P1]
    Lines6[99].X := 236.641; Lines6[99].Z := 272.674; Lines6[99].F := 800; Lines6[99].CMD := 1; Lines6[99].Param := 0; // G1 Linear [Op10 P1]
    Lines7[0].X := 235.691; Lines7[0].Z := 273.844; Lines7[0].F := 800; Lines7[0].CMD := 1; Lines7[0].Param := 0; // G1 Linear [Op10 P1]
    Lines7[1].X := 234.577; Lines7[1].Z := 275.206; Lines7[1].F := 800; Lines7[1].CMD := 1; Lines7[1].Param := 0; // G1 Linear [Op10 P1]
    Lines7[2].X := 233.618; Lines7[2].Z := 276.369; Lines7[2].F := 800; Lines7[2].CMD := 1; Lines7[2].Param := 0; // G1 Linear [Op10 P1]
    Lines7[3].X := 232.494; Lines7[3].Z := 277.723; Lines7[3].F := 800; Lines7[3].CMD := 1; Lines7[3].Param := 0; // G1 Linear [Op10 P1]
    Lines7[4].X := 231.527; Lines7[4].Z := 278.880; Lines7[4].F := 800; Lines7[4].CMD := 1; Lines7[4].Param := 0; // G1 Linear [Op10 P1]
    Lines7[5].X := 230.393; Lines7[5].Z := 280.226; Lines7[5].F := 800; Lines7[5].CMD := 1; Lines7[5].Param := 0; // G1 Linear [Op10 P1]
    Lines7[6].X := 229.417; Lines7[6].Z := 281.377; Lines7[6].F := 800; Lines7[6].CMD := 1; Lines7[6].Param := 0; // G1 Linear [Op10 P1]
    Lines7[7].X := 228.273; Lines7[7].Z := 282.716; Lines7[7].F := 800; Lines7[7].CMD := 1; Lines7[7].Param := 0; // G1 Linear [Op10 P1]
    Lines7[8].X := 227.124; Lines7[8].Z := 284.050; Lines7[8].F := 800; Lines7[8].CMD := 1; Lines7[8].Param := 0; // G1 Linear [Op10 P1]
    Lines7[9].X := 226.135; Lines7[9].Z := 285.191; Lines7[9].F := 800; Lines7[9].CMD := 1; Lines7[9].Param := 0; // G1 Linear [Op10 P1]
    Lines7[10].X := 224.976; Lines7[10].Z := 286.518; Lines7[10].F := 800; Lines7[10].CMD := 1; Lines7[10].Param := 0; // G1 Linear [Op10 P1]
    Lines7[11].X := 223.978; Lines7[11].Z := 287.652; Lines7[11].F := 800; Lines7[11].CMD := 1; Lines7[11].Param := 0; // G1 Linear [Op10 P1]
    Lines7[12].X := 222.976; Lines7[12].Z := 288.784; Lines7[12].F := 800; Lines7[12].CMD := 1; Lines7[12].Param := 0; // G1 Linear [Op10 P1]
    Lines7[13].X := 221.802; Lines7[13].Z := 290.100; Lines7[13].F := 800; Lines7[13].CMD := 1; Lines7[13].Param := 0; // G1 Linear [Op10 P1]
    Lines7[14].X := 220.623; Lines7[14].Z := 291.412; Lines7[14].F := 800; Lines7[14].CMD := 1; Lines7[14].Param := 0; // G1 Linear [Op10 P1]
    Lines7[15].X := 219.608; Lines7[15].Z := 292.533; Lines7[15].F := 800; Lines7[15].CMD := 1; Lines7[15].Param := 0; // G1 Linear [Op10 P1]
    Lines7[16].X := 218.590; Lines7[16].Z := 293.652; Lines7[16].F := 800; Lines7[16].CMD := 1; Lines7[16].Param := 0; // G1 Linear [Op10 P1]
    Lines7[17].X := 217.396; Lines7[17].Z := 294.953; Lines7[17].F := 800; Lines7[17].CMD := 1; Lines7[17].Param := 0; // G1 Linear [Op10 P1]
    Lines7[18].X := 216.197; Lines7[18].Z := 296.250; Lines7[18].F := 800; Lines7[18].CMD := 1; Lines7[18].Param := 0; // G1 Linear [Op10 P1]
    Lines7[19].X := 215.165; Lines7[19].Z := 297.359; Lines7[19].F := 800; Lines7[19].CMD := 1; Lines7[19].Param := 0; // G1 Linear [Op10 P1]
    Lines7[20].X := 213.956; Lines7[20].Z := 298.648; Lines7[20].F := 800; Lines7[20].CMD := 1; Lines7[20].Param := 0; // G1 Linear [Op10 P1]
    Lines7[21].X := 212.741; Lines7[21].Z := 299.934; Lines7[21].F := 800; Lines7[21].CMD := 1; Lines7[21].Param := 0; // G1 Linear [Op10 P1]
    Lines7[22].X := 202.741; Lines7[22].Z := 289.934; Lines7[22].F := 0; Lines7[22].CMD := 0; Lines7[22].Param := 0; // G0 Rapid [Op10 P1]
    Lines7[23].X := 202.741; Lines7[23].Z := 289.934; Lines7[23].F := 0; Lines7[23].CMD := 20; Lines7[23].Param := 80; // Spindle ON 800 RPM [Op10 P1]
    Lines7[24].X := 275.769; Lines7[24].Z := 205.000; Lines7[24].F := 0; Lines7[24].CMD := 0; Lines7[24].Param := 0; // G0 Rapid [Op11 P1]
    Lines7[25].X := 275.721; Lines7[25].Z := 219.432; Lines7[25].F := 800; Lines7[25].CMD := 1; Lines7[25].Param := 0; // G1 Linear [Op11 P1]
    Lines7[26].X := 275.686; Lines7[26].Z := 219.799; Lines7[26].F := 800; Lines7[26].CMD := 1; Lines7[26].Param := 0; // G1 Linear [Op11 P1]
    Lines7[27].X := 275.584; Lines7[27].Z := 220.153; Lines7[27].F := 800; Lines7[27].CMD := 1; Lines7[27].Param := 0; // G1 Linear [Op11 P1]
    Lines7[28].X := 275.419; Lines7[28].Z := 220.482; Lines7[28].F := 800; Lines7[28].CMD := 1; Lines7[28].Param := 0; // G1 Linear [Op11 P1]
    Lines7[29].X := 274.668; Lines7[29].Z := 222.083; Lines7[29].F := 800; Lines7[29].CMD := 1; Lines7[29].Param := 0; // G1 Linear [Op11 P1]
    Lines7[30].X := 274.019; Lines7[30].Z := 223.452; Lines7[30].F := 800; Lines7[30].CMD := 1; Lines7[30].Param := 0; // G1 Linear [Op11 P1]
    Lines7[31].X := 273.365; Lines7[31].Z := 224.818; Lines7[31].F := 800; Lines7[31].CMD := 1; Lines7[31].Param := 0; // G1 Linear [Op11 P1]
    Lines7[32].X := 272.707; Lines7[32].Z := 226.181; Lines7[32].F := 800; Lines7[32].CMD := 1; Lines7[32].Param := 0; // G1 Linear [Op11 P1]
    Lines7[33].X := 272.044; Lines7[33].Z := 227.541; Lines7[33].F := 800; Lines7[33].CMD := 1; Lines7[33].Param := 0; // G1 Linear [Op11 P1]
    Lines7[34].X := 271.265; Lines7[34].Z := 229.124; Lines7[34].F := 800; Lines7[34].CMD := 1; Lines7[34].Param := 0; // G1 Linear [Op11 P1]
    Lines7[35].X := 270.592; Lines7[35].Z := 230.478; Lines7[35].F := 800; Lines7[35].CMD := 1; Lines7[35].Param := 0; // G1 Linear [Op11 P1]
    Lines7[36].X := 269.915; Lines7[36].Z := 231.829; Lines7[36].F := 800; Lines7[36].CMD := 1; Lines7[36].Param := 0; // G1 Linear [Op11 P1]
    Lines7[37].X := 269.232; Lines7[37].Z := 233.177; Lines7[37].F := 800; Lines7[37].CMD := 1; Lines7[37].Param := 0; // G1 Linear [Op11 P1]
    Lines7[38].X := 268.545; Lines7[38].Z := 234.522; Lines7[38].F := 800; Lines7[38].CMD := 1; Lines7[38].Param := 0; // G1 Linear [Op11 P1]
    Lines7[39].X := 267.854; Lines7[39].Z := 235.864; Lines7[39].F := 800; Lines7[39].CMD := 1; Lines7[39].Param := 0; // G1 Linear [Op11 P1]
    Lines7[40].X := 267.041; Lines7[40].Z := 237.426; Lines7[40].F := 800; Lines7[40].CMD := 1; Lines7[40].Param := 0; // G1 Linear [Op11 P1]
    Lines7[41].X := 266.339; Lines7[41].Z := 238.762; Lines7[41].F := 800; Lines7[41].CMD := 1; Lines7[41].Param := 0; // G1 Linear [Op11 P1]
    Lines7[42].X := 265.633; Lines7[42].Z := 240.095; Lines7[42].F := 800; Lines7[42].CMD := 1; Lines7[42].Param := 0; // G1 Linear [Op11 P1]
    Lines7[43].X := 264.922; Lines7[43].Z := 241.425; Lines7[43].F := 800; Lines7[43].CMD := 1; Lines7[43].Param := 0; // G1 Linear [Op11 P1]
    Lines7[44].X := 264.206; Lines7[44].Z := 242.752; Lines7[44].F := 800; Lines7[44].CMD := 1; Lines7[44].Param := 0; // G1 Linear [Op11 P1]
    Lines7[45].X := 263.485; Lines7[45].Z := 244.076; Lines7[45].F := 800; Lines7[45].CMD := 1; Lines7[45].Param := 0; // G1 Linear [Op11 P1]
    Lines7[46].X := 262.760; Lines7[46].Z := 245.397; Lines7[46].F := 800; Lines7[46].CMD := 1; Lines7[46].Param := 0; // G1 Linear [Op11 P1]
    Lines7[47].X := 262.030; Lines7[47].Z := 246.716; Lines7[47].F := 800; Lines7[47].CMD := 1; Lines7[47].Param := 0; // G1 Linear [Op11 P1]
    Lines7[48].X := 261.173; Lines7[48].Z := 248.250; Lines7[48].F := 800; Lines7[48].CMD := 1; Lines7[48].Param := 0; // G1 Linear [Op11 P1]
    Lines7[49].X := 260.433; Lines7[49].Z := 249.562; Lines7[49].F := 800; Lines7[49].CMD := 1; Lines7[49].Param := 0; // G1 Linear [Op11 P1]
    Lines7[50].X := 259.688; Lines7[50].Z := 250.871; Lines7[50].F := 800; Lines7[50].CMD := 1; Lines7[50].Param := 0; // G1 Linear [Op11 P1]
    Lines7[51].X := 258.814; Lines7[51].Z := 252.395; Lines7[51].F := 800; Lines7[51].CMD := 1; Lines7[51].Param := 0; // G1 Linear [Op11 P1]
    Lines7[52].X := 258.059; Lines7[52].Z := 253.698; Lines7[52].F := 800; Lines7[52].CMD := 1; Lines7[52].Param := 0; // G1 Linear [Op11 P1]
    Lines7[53].X := 257.299; Lines7[53].Z := 254.998; Lines7[53].F := 800; Lines7[53].CMD := 1; Lines7[53].Param := 0; // G1 Linear [Op11 P1]
    Lines7[54].X := 256.535; Lines7[54].Z := 256.295; Lines7[54].F := 800; Lines7[54].CMD := 1; Lines7[54].Param := 0; // G1 Linear [Op11 P1]
    Lines7[55].X := 255.766; Lines7[55].Z := 257.589; Lines7[55].F := 800; Lines7[55].CMD := 1; Lines7[55].Param := 0; // G1 Linear [Op11 P1]
    Lines7[56].X := 254.993; Lines7[56].Z := 258.880; Lines7[56].F := 800; Lines7[56].CMD := 1; Lines7[56].Param := 0; // G1 Linear [Op11 P1]
    Lines7[57].X := 254.215; Lines7[57].Z := 260.169; Lines7[57].F := 800; Lines7[57].CMD := 1; Lines7[57].Param := 0; // G1 Linear [Op11 P1]
    Lines7[58].X := 253.432; Lines7[58].Z := 261.454; Lines7[58].F := 800; Lines7[58].CMD := 1; Lines7[58].Param := 0; // G1 Linear [Op11 P1]
    Lines7[59].X := 252.644; Lines7[59].Z := 262.736; Lines7[59].F := 800; Lines7[59].CMD := 1; Lines7[59].Param := 0; // G1 Linear [Op11 P1]
    Lines7[60].X := 251.720; Lines7[60].Z := 264.229; Lines7[60].F := 800; Lines7[60].CMD := 1; Lines7[60].Param := 0; // G1 Linear [Op11 P1]
    Lines7[61].X := 250.922; Lines7[61].Z := 265.505; Lines7[61].F := 800; Lines7[61].CMD := 1; Lines7[61].Param := 0; // G1 Linear [Op11 P1]
    Lines7[62].X := 250.120; Lines7[62].Z := 266.778; Lines7[62].F := 800; Lines7[62].CMD := 1; Lines7[62].Param := 0; // G1 Linear [Op11 P1]
    Lines7[63].X := 249.313; Lines7[63].Z := 268.049; Lines7[63].F := 800; Lines7[63].CMD := 1; Lines7[63].Param := 0; // G1 Linear [Op11 P1]
    Lines7[64].X := 248.501; Lines7[64].Z := 269.316; Lines7[64].F := 800; Lines7[64].CMD := 1; Lines7[64].Param := 0; // G1 Linear [Op11 P1]
    Lines7[65].X := 247.548; Lines7[65].Z := 270.791; Lines7[65].F := 800; Lines7[65].CMD := 1; Lines7[65].Param := 0; // G1 Linear [Op11 P1]
    Lines7[66].X := 246.726; Lines7[66].Z := 272.052; Lines7[66].F := 800; Lines7[66].CMD := 1; Lines7[66].Param := 0; // G1 Linear [Op11 P1]
    Lines7[67].X := 245.900; Lines7[67].Z := 273.310; Lines7[67].F := 800; Lines7[67].CMD := 1; Lines7[67].Param := 0; // G1 Linear [Op11 P1]
    Lines7[68].X := 245.068; Lines7[68].Z := 274.566; Lines7[68].F := 800; Lines7[68].CMD := 1; Lines7[68].Param := 0; // G1 Linear [Op11 P1]
    Lines7[69].X := 244.233; Lines7[69].Z := 275.818; Lines7[69].F := 800; Lines7[69].CMD := 1; Lines7[69].Param := 0; // G1 Linear [Op11 P1]
    Lines7[70].X := 243.392; Lines7[70].Z := 277.068; Lines7[70].F := 800; Lines7[70].CMD := 1; Lines7[70].Param := 0; // G1 Linear [Op11 P1]
    Lines7[71].X := 242.405; Lines7[71].Z := 278.522; Lines7[71].F := 800; Lines7[71].CMD := 1; Lines7[71].Param := 0; // G1 Linear [Op11 P1]
    Lines7[72].X := 241.555; Lines7[72].Z := 279.765; Lines7[72].F := 800; Lines7[72].CMD := 1; Lines7[72].Param := 0; // G1 Linear [Op11 P1]
    Lines7[73].X := 240.699; Lines7[73].Z := 281.005; Lines7[73].F := 800; Lines7[73].CMD := 1; Lines7[73].Param := 0; // G1 Linear [Op11 P1]
    Lines7[74].X := 239.696; Lines7[74].Z := 282.448; Lines7[74].F := 800; Lines7[74].CMD := 1; Lines7[74].Param := 0; // G1 Linear [Op11 P1]
    Lines7[75].X := 238.830; Lines7[75].Z := 283.682; Lines7[75].F := 800; Lines7[75].CMD := 1; Lines7[75].Param := 0; // G1 Linear [Op11 P1]
